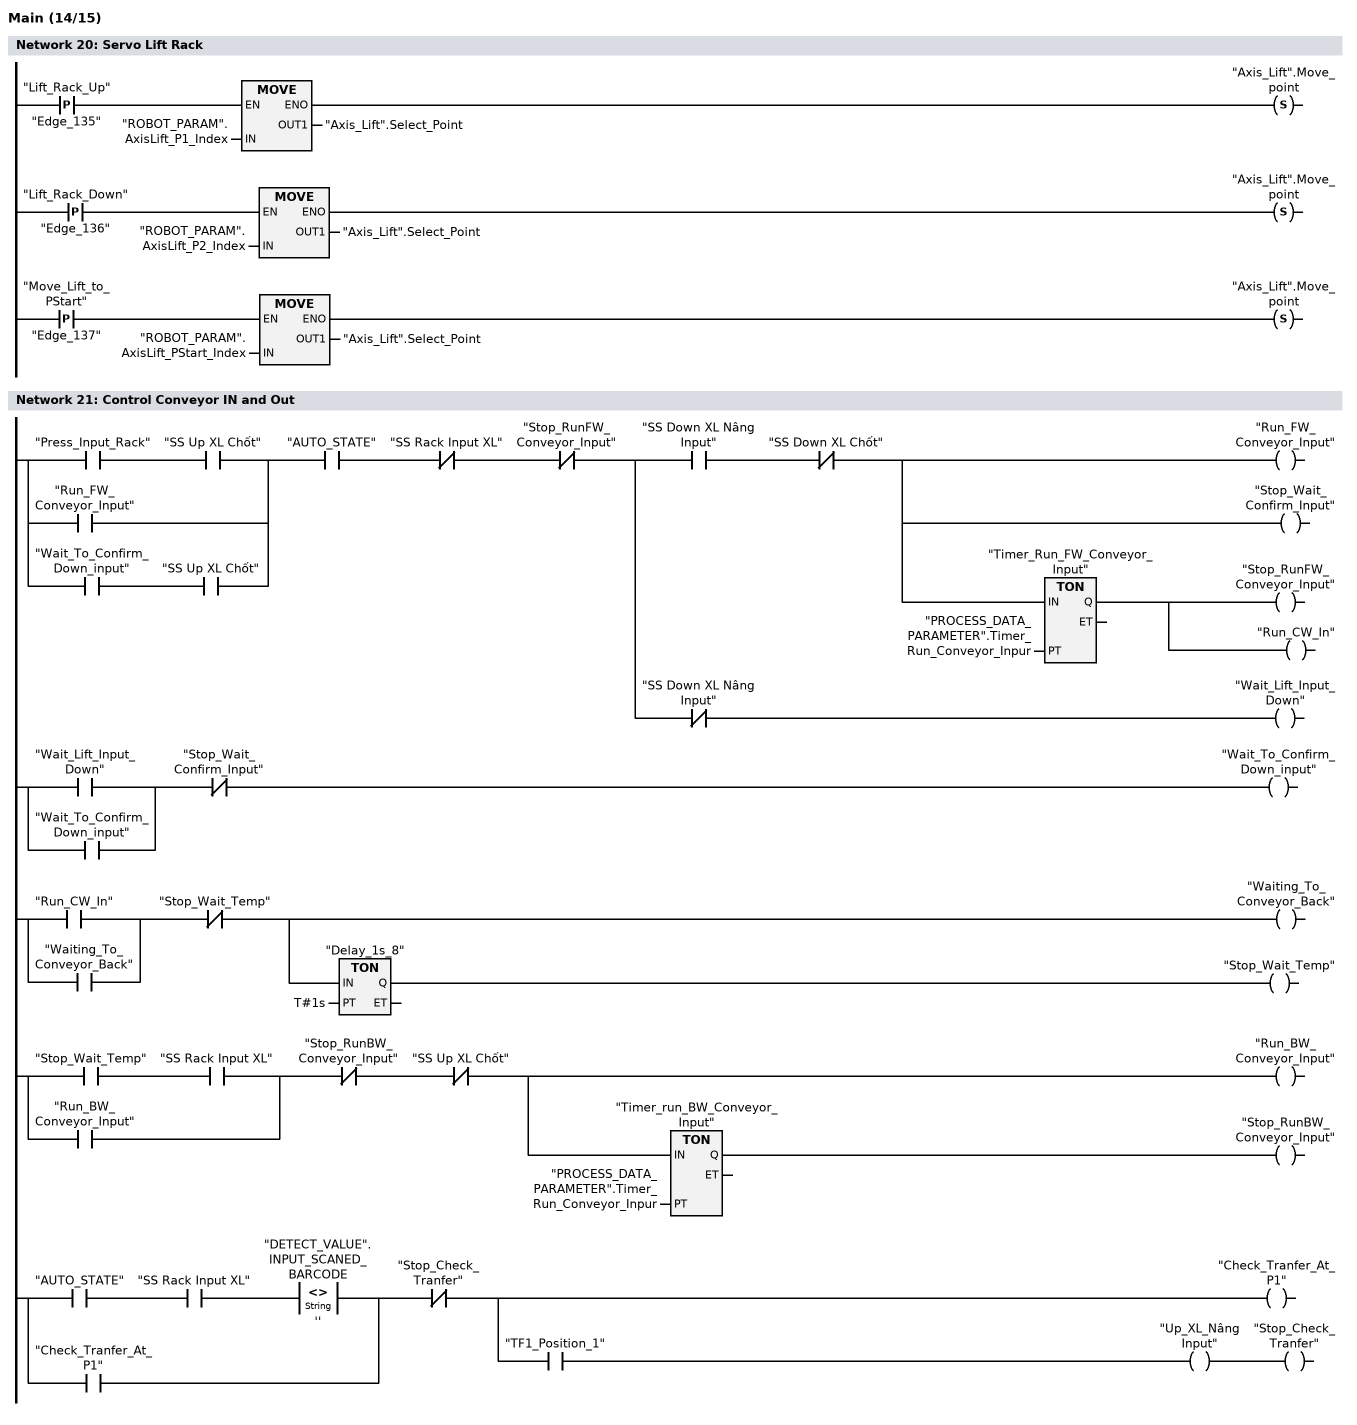
   RUNG wire#powerrail
      P_Contact(operand := "Lift_Rack_Up", bit := "Edge_135")
      { S7_GenerateENO := "TRUE" } Move(in := "ROBOT_PARAM".AxisLift_P1_Index, out1 => "Axis_Lift".Select_Point)
      S_Coil( "Axis_Lift".Move_point )
   END_RUNG
   RUNG wire#powerrail
      P_Contact(operand := "Lift_Rack_Down", bit := "Edge_136")
      { S7_GenerateENO := "TRUE" } Move(in := "ROBOT_PARAM".AxisLift_P2_Index, out1 => "Axis_Lift".Select_Point)
      S_Coil( "Axis_Lift".Move_point )
   END_RUNG
   RUNG wire#powerrail
      P_Contact(operand := "Move_Lift_to_PStart", bit := "Edge_137")
      { S7_GenerateENO := "TRUE" } Move(in := "ROBOT_PARAM".AxisLift_PStart_Index, out1 => "Axis_Lift".Select_Point)
      S_Coil( "Axis_Lift".Move_point )
   END_RUNG
   // the same network as SCL:
   // ENO of a box is taken as its EN; it also drops when the box reports an error
   #_w1 := "Lift_Rack_Up" AND NOT "Edge_135";   // rising edge of "Lift_Rack_Up"
   "Edge_135" := "Lift_Rack_Up";
   IF #_w1 THEN
       "Axis_Lift".Select_Point := "ROBOT_PARAM".AxisLift_P1_Index;
       "Axis_Lift".Move_point := TRUE;
   END_IF;
   #_w2 := "Lift_Rack_Down" AND NOT "Edge_136";   // rising edge of "Lift_Rack_Down"
   "Edge_136" := "Lift_Rack_Down";
   IF #_w2 THEN
       "Axis_Lift".Select_Point := "ROBOT_PARAM".AxisLift_P2_Index;
       "Axis_Lift".Move_point := TRUE;
   END_IF;
   #_w3 := "Move_Lift_to_PStart" AND NOT "Edge_137";   // rising edge of "Move_Lift_to_PStart"
   "Edge_137" := "Move_Lift_to_PStart";
   IF #_w3 THEN
       "Axis_Lift".Select_Point := "ROBOT_PARAM".AxisLift_PStart_Index;
       "Axis_Lift".Move_point := TRUE;
   END_IF;
END_REGION

REGION Network 21: Control Conveyor IN and Out
   #_w1 := (("Press_Input_Rack" AND "SS Up XL Chốt") OR "Run_FW_Conveyor_Input" OR ("Wait_To_Confirm_Down_input" AND "SS Up XL Chốt")) AND "AUTO_STATE" AND NOT "SS Rack Input XL" AND NOT "Stop_RunFW_Conveyor_Input";
   "Run_FW_Conveyor_Input" := #_w1 AND "SS Down XL Nâng Input" AND NOT "SS Down XL Chốt";
   "Stop_Wait_Confirm_Input" := "Run_FW_Conveyor_Input";
   "Timer_Run_FW_Conveyor_Input".TON(IN := "Run_FW_Conveyor_Input",
                           PT := "PROCESS_DATA_PARAMETER".Timer_Run_Conveyor_Inpur);
   "Stop_RunFW_Conveyor_Input" := "Timer_Run_FW_Conveyor_Input".Q;
   "Run_CW_In" := "Timer_Run_FW_Conveyor_Input".Q;
   "Wait_Lift_Input_Down" := #_w1 AND NOT "SS Down XL Nâng Input";
   "Wait_To_Confirm_Down_input" := ("Wait_Lift_Input_Down" OR "Wait_To_Confirm_Down_input") AND NOT "Stop_Wait_Confirm_Input";
   "Waiting_To_Conveyor_Back" := ("Run_CW_In" OR "Waiting_To_Conveyor_Back") AND NOT "Stop_Wait_Temp";
   "Delay_1s_8".TON(IN := "Waiting_To_Conveyor_Back", PT := T#1s);
   "Stop_Wait_Temp" := "Delay_1s_8".Q;
   "Run_BW_Conveyor_Input" := (("Stop_Wait_Temp" AND "SS Rack Input XL") OR "Run_BW_Conveyor_Input") AND NOT "Stop_RunBW_Conveyor_Input" AND NOT "SS Up XL Chốt";
   "Timer_run_BW_Conveyor_Input".TON(IN := "Run_BW_Conveyor_Input",
                           PT := "PROCESS_DATA_PARAMETER".Timer_Run_Conveyor_Inpur);
   "Stop_RunBW_Conveyor_Input" := "Timer_run_BW_Conveyor_Input".Q;
   "Check_Tranfer_At_P1" := (("AUTO_STATE" AND "SS Rack Input XL" AND ("DETECT_VALUE".INPUT_SCANED_BARCODE <> '')) OR "Check_Tranfer_At_P1") AND NOT "Stop_Check_Tranfer";
   "Up_XL_Nâng Input" := "Check_Tranfer_At_P1" AND "TF1_Position_1";
   "Stop_Check_Tranfer" := "Up_XL_Nâng Input";
END_REGION

REGION Network 22: Conveyor Out
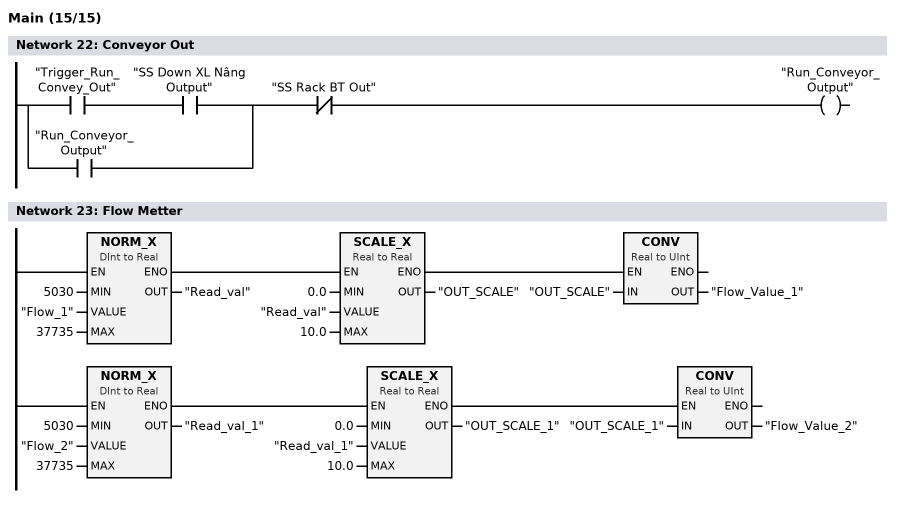
   RUNG wire#powerrail
      Contact( "Trigger_Run_Convey_Out" )
      Contact( "SS Down XL Nâng Output" )
      wire#w1
      I_Contact( "SS Rack BT Out" )
      Coil( "Run_Conveyor_Output" )
   END_RUNG
   RUNG wire#powerrail
      Contact( "Run_Conveyor_Output" )
   END_RUNG wire#w1
   // the same network as SCL:
   "Run_Conveyor_Output" := (("Trigger_Run_Convey_Out" AND "SS Down XL Nâng Output") OR "Run_Conveyor_Output") AND NOT "SS Rack BT Out";
END_REGION

REGION Network 23: Flow Metter
   RUNG wire#powerrail
      { S7_Templates := "[SrcType := DInt, DestType := Real]"; S7_GenerateENO := "TRUE" } Normalize(min := 5030, value := "Flow_1", max := 37735, out => "Read_val")
      { S7_Templates := "[SrcType := Real, DestType := Real]"; S7_GenerateENO := "TRUE" } Scale(min := 0.0, value := "Read_val", max := 10.0, out => "OUT_SCALE")
      { S7_Templates := "[SrcType := Real, DestType := UInt]"; S7_GenerateENO := "TRUE" } Convert(in := "OUT_SCALE", out => "Flow_Value_1")
   END_RUNG
   RUNG wire#powerrail
      { S7_Templates := "[SrcType := DInt, DestType := Real]"; S7_GenerateENO := "TRUE" } Normalize(min := 5030, value := "Flow_2", max := 37735, out => "Read_val_1")
      { S7_Templates := "[SrcType := Real, DestType := Real]"; S7_GenerateENO := "TRUE" } Scale(min := 0.0, value := "Read_val_1", max := 10.0, out => "OUT_SCALE_1")
      { S7_Templates := "[SrcType := Real, DestType := UInt]"; S7_GenerateENO := "TRUE" } Convert(in := "OUT_SCALE_1", out => "Flow_Value_2")
   END_RUNG
   // the same network as SCL:
   // ENO of a box is taken as its EN; it also drops when the box reports an error
   "Read_val" := NORM_X(MIN := 5030, VALUE := "Flow_1", MAX := 37735);
   "OUT_SCALE" := SCALE_X(MIN := 0.0, VALUE := "Read_val", MAX := 10.0);
   "Flow_Value_1" := REAL_TO_UINT("OUT_SCALE");
   "Read_val_1" := NORM_X(MIN := 5030, VALUE := "Flow_2", MAX := 37735);
   "OUT_SCALE_1" := SCALE_X(MIN := 0.0, VALUE := "Read_val_1", MAX := 10.0);
   "Flow_Value_2" := REAL_TO_UINT("OUT_SCALE_1");
END_REGION
END_ORGANIZATION_BLOCK

ORGANIZATION_BLOCK "MOTOR_CONTROL"   // OB123, LAD, ProgramCycle
TITLE = "Main Program Sweep (Cycle)"
{ S7_Optimized_Access := 'TRUE' }
VERSION : 0.1
   VAR_INPUT
      Initial_Call : Bool;   // Initial call of this OB
      Remanence : Bool;   // =True, if remanent data are available
   END_VAR
   VAR_TEMP   // added for the SCL form of the ladder/FBD networks
      _w1 : Bool;
      _w2 : Bool;
      _w3 : Bool;
      _w4 : Bool;
      _w5 : Bool;
      _w6 : Bool;
      _w7 : Bool;
      _w8 : Bool;
      _w9 : Bool;
      _w10 : Bool;
      _w11 : Bool;
      _w12 : Bool;
      _w13 : Bool;
      _w14 : Bool;
      _w15 : Bool;
      _w16 : Bool;
      _w17 : Bool;
      _w18 : Bool;
      _w19 : Bool;
      _w20 : Bool;
      _w21 : Bool;
      _w22 : Bool;
      _w23 : Bool;
      _w24 : Bool;
      _w25 : Bool;
      _w26 : Bool;
      _w27 : Bool;
      _w28 : Bool;
      _w29 : Bool;
      _w30 : Bool;
      _w31 : Bool;
      _w32 : Bool;
      _w33 : Bool;
      _w34 : Bool;
      _w35 : Bool;
      _w36 : Bool;
      _w37 : Bool;
      _w38 : Bool;
      _w39 : Bool;
      _w40 : Bool;
   END_VAR
BEGIN

REGION Network 1: MODBUS INITIALIZE
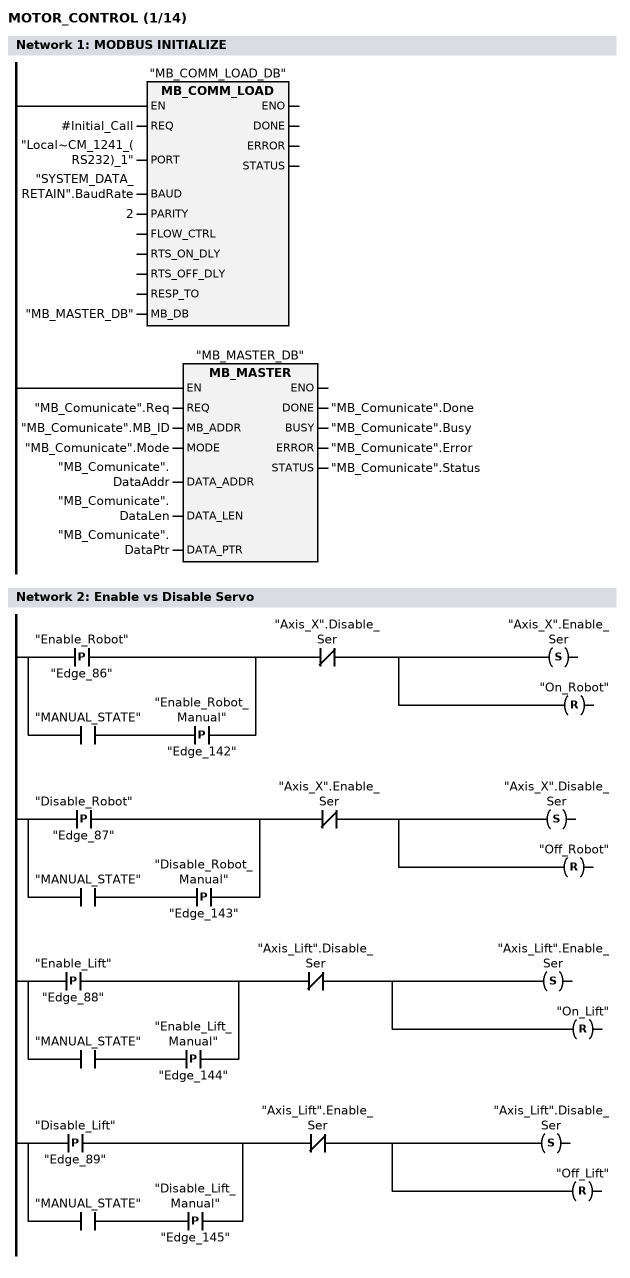
   "MB_COMM_LOAD_DB"(REQ := #Initial_Call,   // MB_COMM_LOAD
                     PORT := "Local~CM_1241_(RS232)_1",
                     BAUD := "SYSTEM_DATA_RETAIN".BaudRate,
                     PARITY := 2,
                     MB_DB := "MB_MASTER_DB");
   "MB_MASTER_DB"(REQ := "MB_Comunicate".Req,   // MB_MASTER
                  MB_ADDR := "MB_Comunicate".MB_ID,
                  MODE := "MB_Comunicate".Mode,
                  DATA_ADDR := "MB_Comunicate".DataAddr,
                  DATA_LEN := "MB_Comunicate".DataLen,
                  DATA_PTR := "MB_Comunicate".DataPtr,
                  DONE => "MB_Comunicate".Done,
                  BUSY => "MB_Comunicate".Busy,
                  ERROR => "MB_Comunicate".Error,
                  STATUS => "MB_Comunicate".Status);
END_REGION

REGION Network 2: Enable vs Disable Servo
   RUNG wire#powerrail
      P_Contact(operand := "Enable_Robot", bit := "Edge_86")
      wire#w1
      I_Contact( "Axis_X".Disable_Ser )
      wire#w2
      S_Coil( "Axis_X".Enable_Ser )
   END_RUNG
   RUNG wire#powerrail
      Contact( "MANUAL_STATE" )
      P_Contact(operand := "Enable_Robot_Manual", bit := "Edge_142")
   END_RUNG wire#w1
   RUNG wire#w2
      R_Coil( "On_Robot" )
   END_RUNG
   RUNG wire#powerrail
      P_Contact(operand := "Disable_Robot", bit := "Edge_87")
      wire#w3
      I_Contact( "Axis_X".Enable_Ser )
      wire#w4
      S_Coil( "Axis_X".Disable_Ser )
   END_RUNG
   RUNG wire#powerrail
      Contact( "MANUAL_STATE" )
      P_Contact(operand := "Disable_Robot_Manual", bit := "Edge_143")
   END_RUNG wire#w3
   RUNG wire#w4
      R_Coil( "Off_Robot" )
   END_RUNG
   RUNG wire#powerrail
      P_Contact(operand := "Enable_Lift", bit := "Edge_88")
      wire#w5
      I_Contact( "Axis_Lift".Disable_Ser )
      wire#w6
      S_Coil( "Axis_Lift".Enable_Ser )
   END_RUNG
   RUNG wire#powerrail
      Contact( "MANUAL_STATE" )
      P_Contact(operand := "Enable_Lift_Manual", bit := "Edge_144")
   END_RUNG wire#w5
   RUNG wire#w6
      R_Coil( "On_Lift" )
   END_RUNG
   RUNG wire#powerrail
      P_Contact(operand := "Disable_Lift", bit := "Edge_89")
      wire#w7
      I_Contact( "Axis_Lift".Enable_Ser )
      wire#w8
      S_Coil( "Axis_Lift".Disable_Ser )
   END_RUNG
   RUNG wire#powerrail
      Contact( "MANUAL_STATE" )
      P_Contact(operand := "Disable_Lift_Manual", bit := "Edge_145")
   END_RUNG wire#w7
   RUNG wire#w8
      R_Coil( "Off_Lift" )
   END_RUNG
   // the same network as SCL:
   #_w1 := "Enable_Robot" AND NOT "Edge_86";   // rising edge of "Enable_Robot"
   "Edge_86" := "Enable_Robot";
   #_w2 := "MANUAL_STATE" AND "Enable_Robot_Manual" AND NOT "Edge_142";   // rising edge of "Enable_Robot_Manual"
   "Edge_142" := "Enable_Robot_Manual";
   IF (#_w1 OR #_w2) AND NOT "Axis_X".Disable_Ser THEN
       "Axis_X".Enable_Ser := TRUE;
       "On_Robot" := FALSE;
   END_IF;
   #_w3 := "Disable_Robot" AND NOT "Edge_87";   // rising edge of "Disable_Robot"
   "Edge_87" := "Disable_Robot";
   #_w4 := "MANUAL_STATE" AND "Disable_Robot_Manual" AND NOT "Edge_143";   // rising edge of "Disable_Robot_Manual"
   "Edge_143" := "Disable_Robot_Manual";
   IF (#_w3 OR #_w4) AND NOT "Axis_X".Enable_Ser THEN
       "Axis_X".Disable_Ser := TRUE;
       "Off_Robot" := FALSE;
   END_IF;
   #_w5 := "Enable_Lift" AND NOT "Edge_88";   // rising edge of "Enable_Lift"
   "Edge_88" := "Enable_Lift";
   #_w6 := "MANUAL_STATE" AND "Enable_Lift_Manual" AND NOT "Edge_144";   // rising edge of "Enable_Lift_Manual"
   "Edge_144" := "Enable_Lift_Manual";
   IF (#_w5 OR #_w6) AND NOT "Axis_Lift".Disable_Ser THEN
       "Axis_Lift".Enable_Ser := TRUE;
       "On_Lift" := FALSE;
   END_IF;
   #_w7 := "Disable_Lift" AND NOT "Edge_89";   // rising edge of "Disable_Lift"
   "Edge_89" := "Disable_Lift";
   #_w8 := "MANUAL_STATE" AND "Disable_Lift_Manual" AND NOT "Edge_145";   // rising edge of "Disable_Lift_Manual"
   "Edge_145" := "Disable_Lift_Manual";
   IF (#_w7 OR #_w8) AND NOT "Axis_Lift".Enable_Ser THEN
       "Axis_Lift".Disable_Ser := TRUE;
       "Off_Lift" := FALSE;
   END_IF;
END_REGION

REGION Network 3: AXIS X
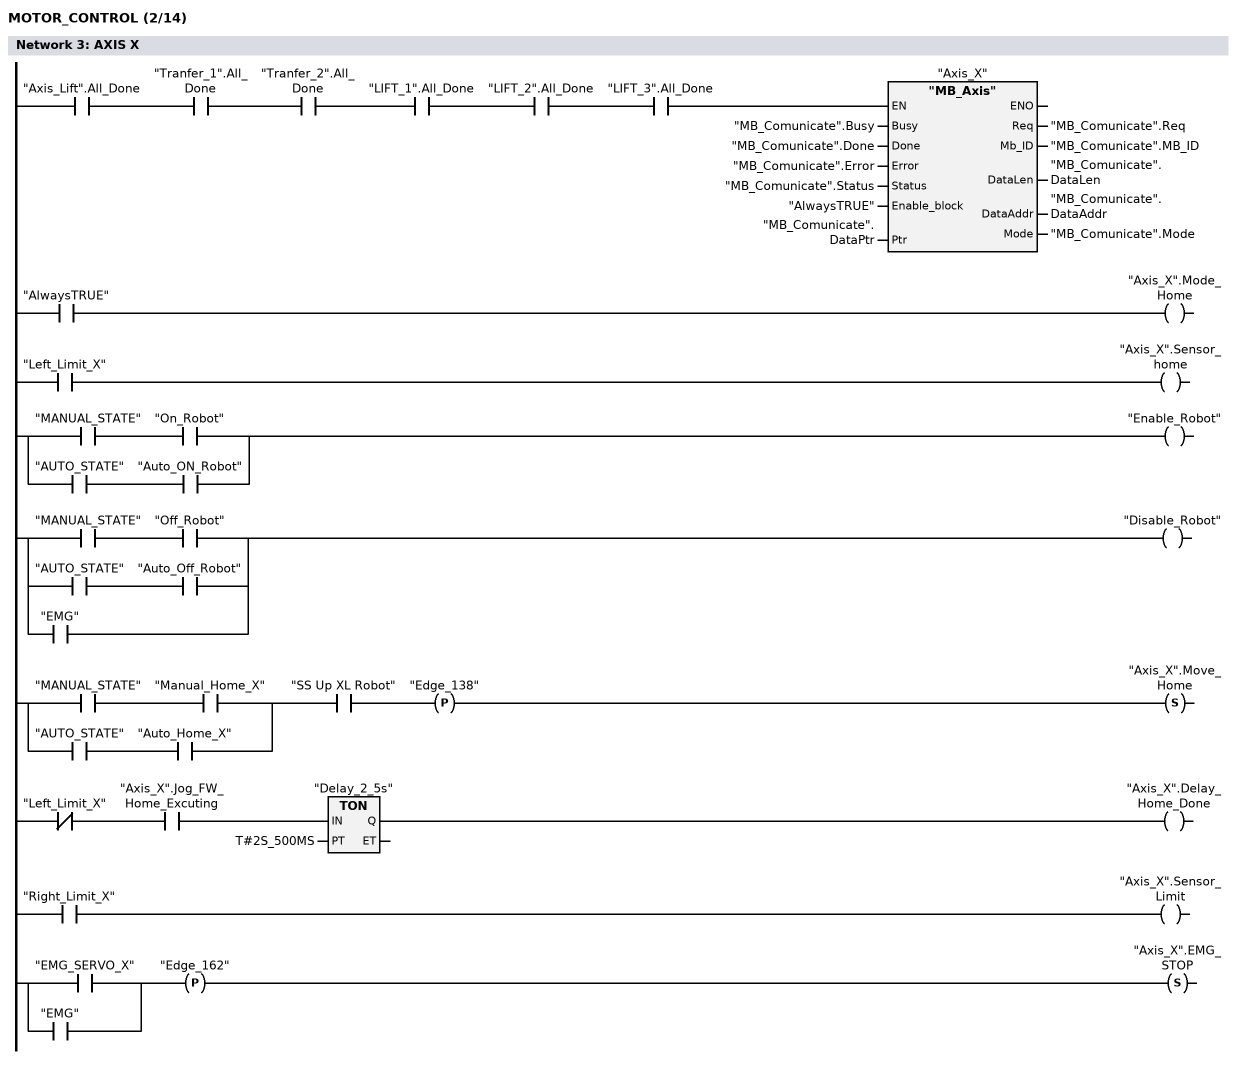
   IF "Axis_Lift".All_Done AND "Tranfer_1".All_Done AND "Tranfer_2".All_Done AND "LIFT_1".All_Done AND "LIFT_2".All_Done AND "LIFT_3".All_Done THEN
       "Axis_X"(Busy := "MB_Comunicate".Busy,   // "MB_Axis"
                Done := "MB_Comunicate".Done,
                Error := "MB_Comunicate".Error,
                Status := "MB_Comunicate".Status,
                Enable_block := "AlwaysTRUE",
                Ptr := "MB_Comunicate".DataPtr,
                Req => "MB_Comunicate".Req,
                Mb_ID => "MB_Comunicate".MB_ID,
                DataLen => "MB_Comunicate".DataLen,
                DataAddr => "MB_Comunicate".DataAddr,
                Mode => "MB_Comunicate".Mode);
   END_IF;
   "Axis_X".Mode_Home := "AlwaysTRUE";
   "Axis_X".Sensor_home := "Left_Limit_X";
   "Enable_Robot" := ("MANUAL_STATE" AND "On_Robot") OR ("AUTO_STATE" AND "Auto_ON_Robot");
   "Disable_Robot" := ("MANUAL_STATE" AND "Off_Robot") OR ("AUTO_STATE" AND "Auto_Off_Robot") OR "EMG";
   #_w1 := (("MANUAL_STATE" AND "Manual_Home_X") OR ("AUTO_STATE" AND "Auto_Home_X")) AND "SS Up XL Robot";
   #_w2 := #_w1 AND NOT "Edge_138";   // rising edge
   "Edge_138" := #_w1;
   IF #_w2 THEN "Axis_X".Move_Home := TRUE; END_IF;
   "Delay_2_5s".TON(IN := NOT "Left_Limit_X" AND "Axis_X".Jog_FW_Home_Excuting, PT := T#2S_500MS);
   "Axis_X".Delay_Home_Done := "Delay_2_5s".Q;
   "Axis_X".Sensor_Limit := "Right_Limit_X";
   #_w3 := "EMG_SERVO_X" OR "EMG";
   #_w4 := #_w3 AND NOT "Edge_162";   // rising edge
   "Edge_162" := #_w3;
   IF #_w4 THEN "Axis_X".EMG_STOP := TRUE; END_IF;
END_REGION

REGION Network 4: AXIS LIFT
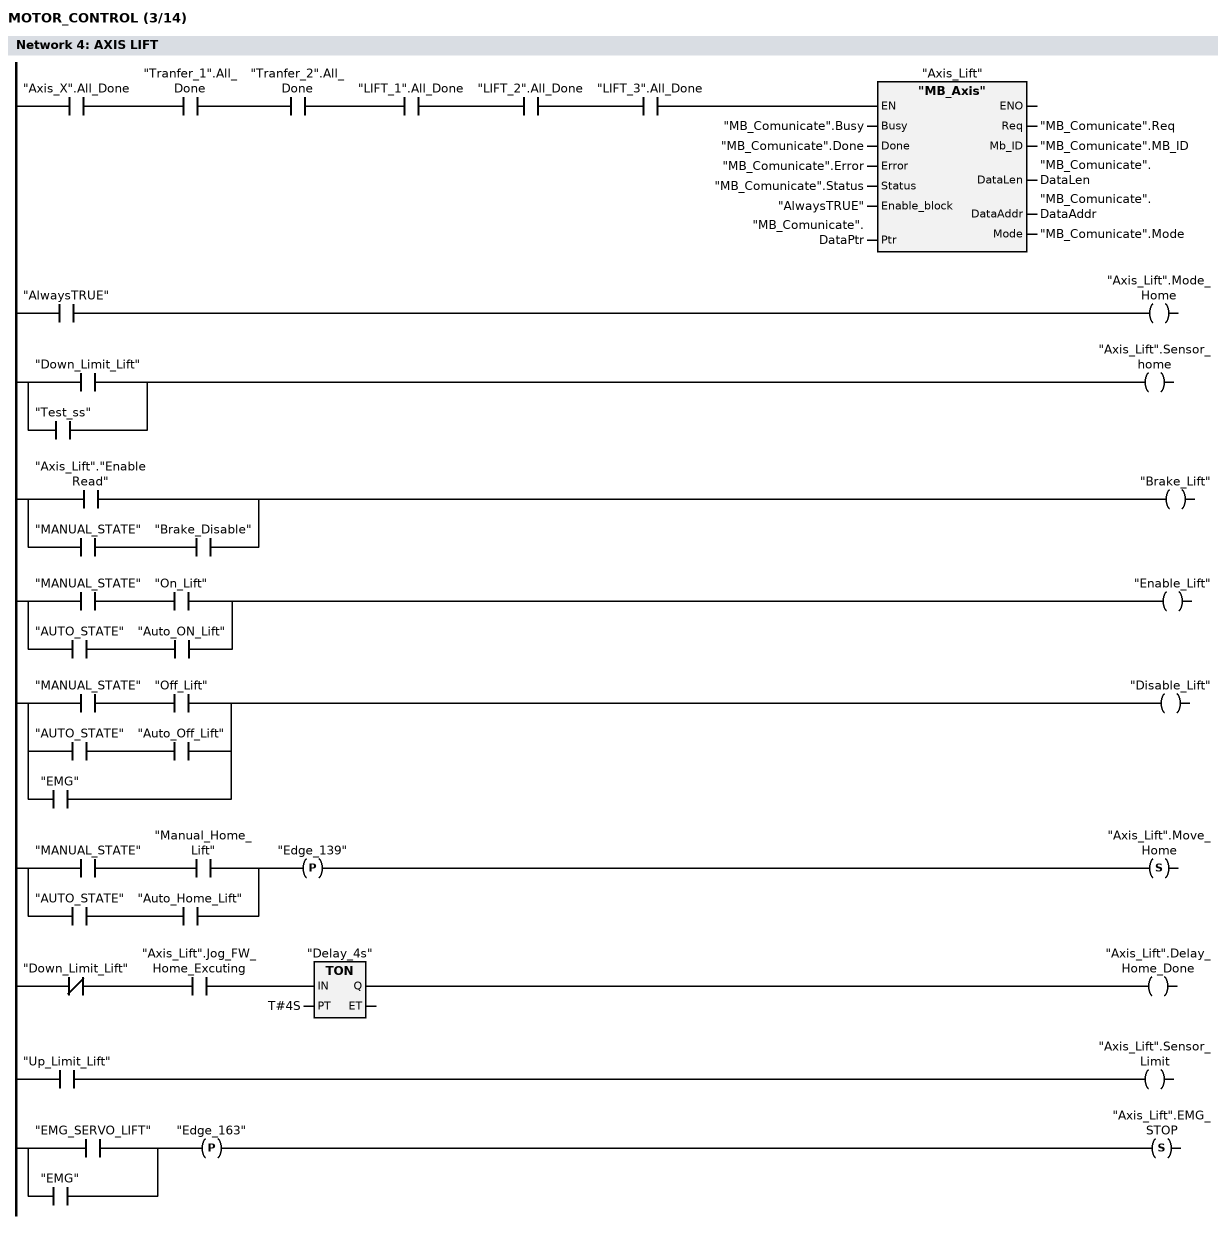
   IF "Axis_X".All_Done AND "Tranfer_1".All_Done AND "Tranfer_2".All_Done AND "LIFT_1".All_Done AND "LIFT_2".All_Done AND "LIFT_3".All_Done THEN
       "Axis_Lift"(Busy := "MB_Comunicate".Busy,   // "MB_Axis"
                   Done := "MB_Comunicate".Done,
                   Error := "MB_Comunicate".Error,
                   Status := "MB_Comunicate".Status,
                   Enable_block := "AlwaysTRUE",
                   Ptr := "MB_Comunicate".DataPtr,
                   Req => "MB_Comunicate".Req,
                   Mb_ID => "MB_Comunicate".MB_ID,
                   DataLen => "MB_Comunicate".DataLen,
                   DataAddr => "MB_Comunicate".DataAddr,
                   Mode => "MB_Comunicate".Mode);
   END_IF;
   "Axis_Lift".Mode_Home := "AlwaysTRUE";
   "Axis_Lift".Sensor_home := "Down_Limit_Lift" OR "Test_ss";
   "Brake_Lift" := "Axis_Lift"."Enable Read" OR ("MANUAL_STATE" AND "Brake_Disable");
   "Enable_Lift" := ("MANUAL_STATE" AND "On_Lift") OR ("AUTO_STATE" AND "Auto_ON_Lift");
   "Disable_Lift" := ("MANUAL_STATE" AND "Off_Lift") OR ("AUTO_STATE" AND "Auto_Off_Lift") OR "EMG";
   #_w1 := ("MANUAL_STATE" AND "Manual_Home_Lift") OR ("AUTO_STATE" AND "Auto_Home_Lift");
   #_w2 := #_w1 AND NOT "Edge_139";   // rising edge
   "Edge_139" := #_w1;
   IF #_w2 THEN "Axis_Lift".Move_Home := TRUE; END_IF;
   "Delay_4s".TON(IN := NOT "Down_Limit_Lift" AND "Axis_Lift".Jog_FW_Home_Excuting, PT := T#4S);
   "Axis_Lift".Delay_Home_Done := "Delay_4s".Q;
   "Axis_Lift".Sensor_Limit := "Up_Limit_Lift";
   #_w3 := "EMG_SERVO_LIFT" OR "EMG";
   #_w4 := #_w3 AND NOT "Edge_163";   // rising edge
   "Edge_163" := #_w3;
   IF #_w4 THEN "Axis_Lift".EMG_STOP := TRUE; END_IF;
END_REGION

REGION Network 5: Data Position
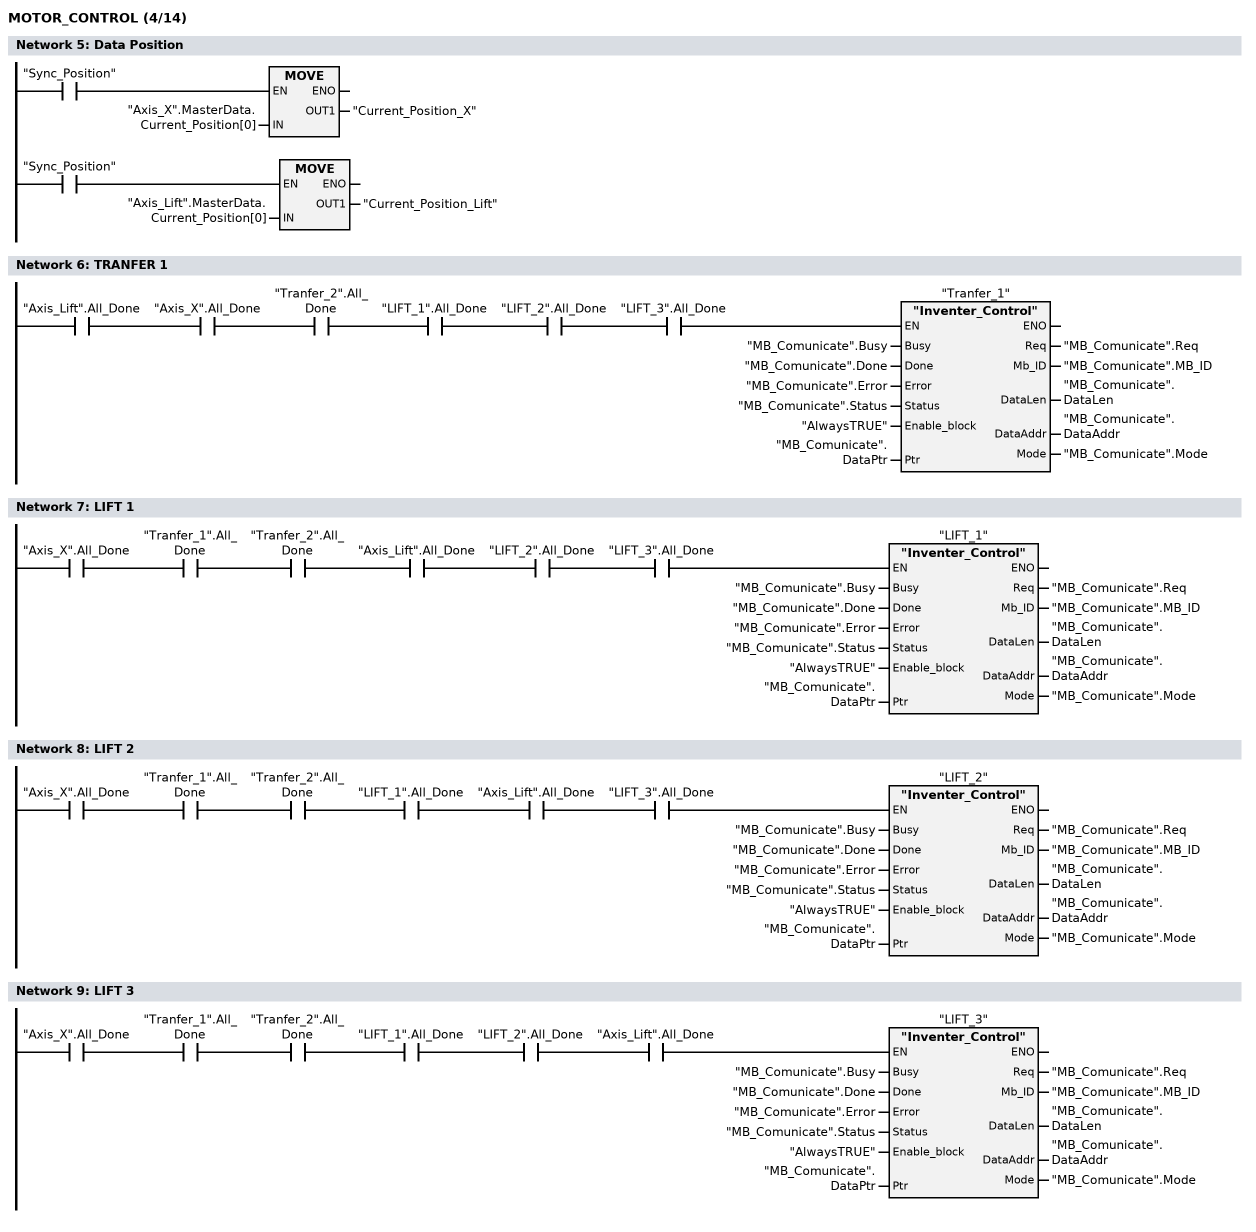
   RUNG wire#powerrail
      Contact( "Sync_Position" )
      { S7_GenerateENO := "TRUE" } Move(in := "Axis_X".MasterData.Current_Position[0], out1 => "Current_Position_X")
   END_RUNG
   RUNG wire#powerrail
      Contact( "Sync_Position" )
      { S7_GenerateENO := "TRUE" } Move(in := "Axis_Lift".MasterData.Current_Position[0], out1 => "Current_Position_Lift")
   END_RUNG
   // the same network as SCL:
   IF "Sync_Position" THEN
       "Current_Position_X" := "Axis_X".MasterData.Current_Position[0];
       "Current_Position_Lift" := "Axis_Lift".MasterData.Current_Position[0];
   END_IF;
END_REGION

REGION Network 6: TRANFER 1
   RUNG wire#powerrail
      Contact( "Axis_Lift".All_Done )
      Contact( "Axis_X".All_Done )
      Contact( "Tranfer_2".All_Done )
      Contact( "LIFT_1".All_Done )
      Contact( "LIFT_2".All_Done )
      Contact( "LIFT_3".All_Done )
      "Tranfer_1"(Busy := "MB_Comunicate".Busy, Done := "MB_Comunicate".Done, Error := "MB_Comunicate".Error, Status := "MB_Comunicate".Status, Enable_block := "AlwaysTRUE", Ptr := "MB_Comunicate".DataPtr, Req => "MB_Comunicate".Req, Mb_ID => "MB_Comunicate".MB_ID, DataLen => "MB_Comunicate".DataLen, DataAddr => "MB_Comunicate".DataAddr, Mode => "MB_Comunicate".Mode)
   END_RUNG
   // the same network as SCL:
   IF "Axis_Lift".All_Done AND "Axis_X".All_Done AND "Tranfer_2".All_Done AND "LIFT_1".All_Done AND "LIFT_2".All_Done AND "LIFT_3".All_Done THEN
       "Tranfer_1"(Busy := "MB_Comunicate".Busy,   // "Inventer_Control"
                   Done := "MB_Comunicate".Done,
                   Error := "MB_Comunicate".Error,
                   Status := "MB_Comunicate".Status,
                   Enable_block := "AlwaysTRUE",
                   Ptr := "MB_Comunicate".DataPtr,
                   Req => "MB_Comunicate".Req,
                   Mb_ID => "MB_Comunicate".MB_ID,
                   DataLen => "MB_Comunicate".DataLen,
                   DataAddr => "MB_Comunicate".DataAddr,
                   Mode => "MB_Comunicate".Mode);
   END_IF;
END_REGION

REGION Network 7: LIFT 1
   RUNG wire#powerrail
      Contact( "Axis_X".All_Done )
      Contact( "Tranfer_1".All_Done )
      Contact( "Tranfer_2".All_Done )
      Contact( "Axis_Lift".All_Done )
      Contact( "LIFT_2".All_Done )
      Contact( "LIFT_3".All_Done )
      "LIFT_1"(Busy := "MB_Comunicate".Busy, Done := "MB_Comunicate".Done, Error := "MB_Comunicate".Error, Status := "MB_Comunicate".Status, Enable_block := "AlwaysTRUE", Ptr := "MB_Comunicate".DataPtr, Req => "MB_Comunicate".Req, Mb_ID => "MB_Comunicate".MB_ID, DataLen => "MB_Comunicate".DataLen, DataAddr => "MB_Comunicate".DataAddr, Mode => "MB_Comunicate".Mode)
   END_RUNG
   // the same network as SCL:
   IF "Axis_X".All_Done AND "Tranfer_1".All_Done AND "Tranfer_2".All_Done AND "Axis_Lift".All_Done AND "LIFT_2".All_Done AND "LIFT_3".All_Done THEN
       "LIFT_1"(Busy := "MB_Comunicate".Busy,   // "Inventer_Control"
                Done := "MB_Comunicate".Done,
                Error := "MB_Comunicate".Error,
                Status := "MB_Comunicate".Status,
                Enable_block := "AlwaysTRUE",
                Ptr := "MB_Comunicate".DataPtr,
                Req => "MB_Comunicate".Req,
                Mb_ID => "MB_Comunicate".MB_ID,
                DataLen => "MB_Comunicate".DataLen,
                DataAddr => "MB_Comunicate".DataAddr,
                Mode => "MB_Comunicate".Mode);
   END_IF;
END_REGION

REGION Network 8: LIFT 2
   RUNG wire#powerrail
      Contact( "Axis_X".All_Done )
      Contact( "Tranfer_1".All_Done )
      Contact( "Tranfer_2".All_Done )
      Contact( "LIFT_1".All_Done )
      Contact( "Axis_Lift".All_Done )
      Contact( "LIFT_3".All_Done )
      "LIFT_2"(Busy := "MB_Comunicate".Busy, Done := "MB_Comunicate".Done, Error := "MB_Comunicate".Error, Status := "MB_Comunicate".Status, Enable_block := "AlwaysTRUE", Ptr := "MB_Comunicate".DataPtr, Req => "MB_Comunicate".Req, Mb_ID => "MB_Comunicate".MB_ID, DataLen => "MB_Comunicate".DataLen, DataAddr => "MB_Comunicate".DataAddr, Mode => "MB_Comunicate".Mode)
   END_RUNG
   // the same network as SCL:
   IF "Axis_X".All_Done AND "Tranfer_1".All_Done AND "Tranfer_2".All_Done AND "LIFT_1".All_Done AND "Axis_Lift".All_Done AND "LIFT_3".All_Done THEN
       "LIFT_2"(Busy := "MB_Comunicate".Busy,   // "Inventer_Control"
                Done := "MB_Comunicate".Done,
                Error := "MB_Comunicate".Error,
                Status := "MB_Comunicate".Status,
                Enable_block := "AlwaysTRUE",
                Ptr := "MB_Comunicate".DataPtr,
                Req => "MB_Comunicate".Req,
                Mb_ID => "MB_Comunicate".MB_ID,
                DataLen => "MB_Comunicate".DataLen,
                DataAddr => "MB_Comunicate".DataAddr,
                Mode => "MB_Comunicate".Mode);
   END_IF;
END_REGION

REGION Network 9: LIFT 3
   RUNG wire#powerrail
      Contact( "Axis_X".All_Done )
      Contact( "Tranfer_1".All_Done )
      Contact( "Tranfer_2".All_Done )
      Contact( "LIFT_1".All_Done )
      Contact( "LIFT_2".All_Done )
      Contact( "Axis_Lift".All_Done )
      "LIFT_3"(Busy := "MB_Comunicate".Busy, Done := "MB_Comunicate".Done, Error := "MB_Comunicate".Error, Status := "MB_Comunicate".Status, Enable_block := "AlwaysTRUE", Ptr := "MB_Comunicate".DataPtr, Req => "MB_Comunicate".Req, Mb_ID => "MB_Comunicate".MB_ID, DataLen => "MB_Comunicate".DataLen, DataAddr => "MB_Comunicate".DataAddr, Mode => "MB_Comunicate".Mode)
   END_RUNG
   // the same network as SCL:
   IF "Axis_X".All_Done AND "Tranfer_1".All_Done AND "Tranfer_2".All_Done AND "LIFT_1".All_Done AND "LIFT_2".All_Done AND "Axis_Lift".All_Done THEN
       "LIFT_3"(Busy := "MB_Comunicate".Busy,   // "Inventer_Control"
                Done := "MB_Comunicate".Done,
                Error := "MB_Comunicate".Error,
                Status := "MB_Comunicate".Status,
                Enable_block := "AlwaysTRUE",
                Ptr := "MB_Comunicate".DataPtr,
                Req => "MB_Comunicate".Req,
                Mb_ID => "MB_Comunicate".MB_ID,
                DataLen => "MB_Comunicate".DataLen,
                DataAddr => "MB_Comunicate".DataAddr,
                Mode => "MB_Comunicate".Mode);
   END_IF;
END_REGION

REGION Network 10
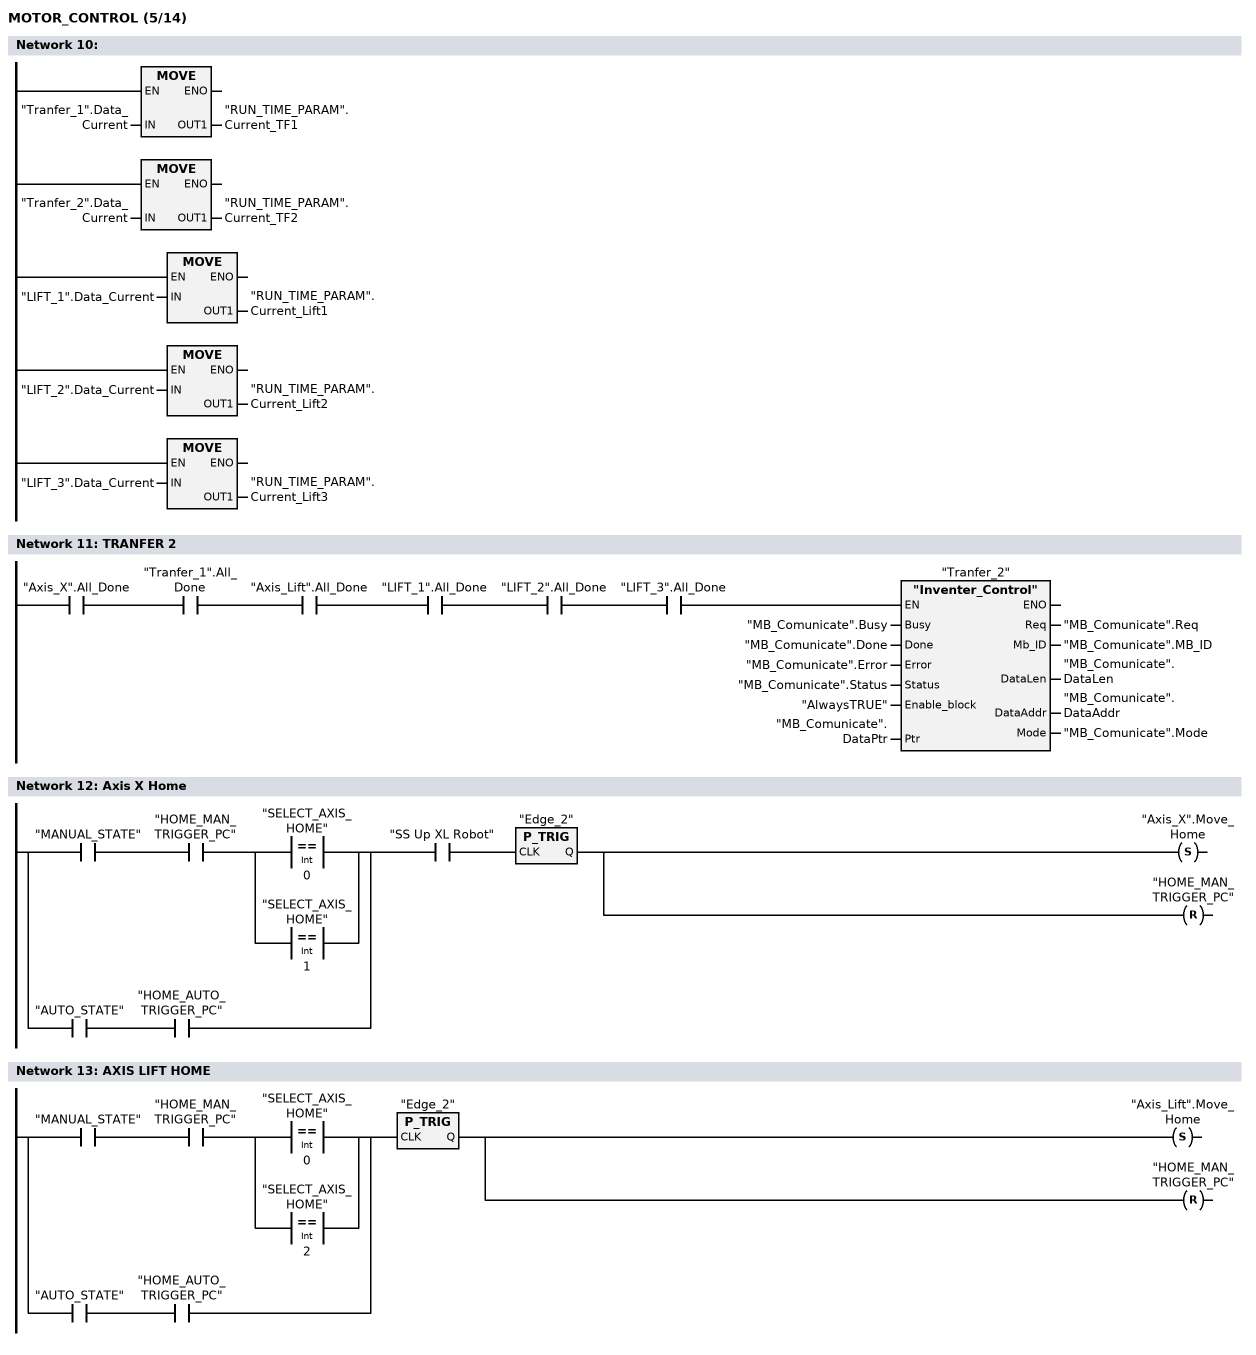
   RUNG wire#powerrail
      { S7_GenerateENO := "TRUE" } Move(in := "Tranfer_1".Data_Current, out1 => "RUN_TIME_PARAM".Current_TF1)
   END_RUNG
   RUNG wire#powerrail
      { S7_GenerateENO := "TRUE" } Move(in := "Tranfer_2".Data_Current, out1 => "RUN_TIME_PARAM".Current_TF2)
   END_RUNG
   RUNG wire#powerrail
      { S7_GenerateENO := "TRUE" } Move(in := "LIFT_1".Data_Current, out1 => "RUN_TIME_PARAM".Current_Lift1)
   END_RUNG
   RUNG wire#powerrail
      { S7_GenerateENO := "TRUE" } Move(in := "LIFT_2".Data_Current, out1 => "RUN_TIME_PARAM".Current_Lift2)
   END_RUNG
   RUNG wire#powerrail
      { S7_GenerateENO := "TRUE" } Move(in := "LIFT_3".Data_Current, out1 => "RUN_TIME_PARAM".Current_Lift3)
   END_RUNG
   // the same network as SCL:
   "RUN_TIME_PARAM".Current_TF1 := "Tranfer_1".Data_Current;
   "RUN_TIME_PARAM".Current_TF2 := "Tranfer_2".Data_Current;
   "RUN_TIME_PARAM".Current_Lift1 := "LIFT_1".Data_Current;
   "RUN_TIME_PARAM".Current_Lift2 := "LIFT_2".Data_Current;
   "RUN_TIME_PARAM".Current_Lift3 := "LIFT_3".Data_Current;
END_REGION

REGION Network 11: TRANFER 2
   RUNG wire#powerrail
      Contact( "Axis_X".All_Done )
      Contact( "Tranfer_1".All_Done )
      Contact( "Axis_Lift".All_Done )
      Contact( "LIFT_1".All_Done )
      Contact( "LIFT_2".All_Done )
      Contact( "LIFT_3".All_Done )
      "Tranfer_2"(Busy := "MB_Comunicate".Busy, Done := "MB_Comunicate".Done, Error := "MB_Comunicate".Error, Status := "MB_Comunicate".Status, Enable_block := "AlwaysTRUE", Ptr := "MB_Comunicate".DataPtr, Req => "MB_Comunicate".Req, Mb_ID => "MB_Comunicate".MB_ID, DataLen => "MB_Comunicate".DataLen, DataAddr => "MB_Comunicate".DataAddr, Mode => "MB_Comunicate".Mode)
   END_RUNG
   // the same network as SCL:
   IF "Axis_X".All_Done AND "Tranfer_1".All_Done AND "Axis_Lift".All_Done AND "LIFT_1".All_Done AND "LIFT_2".All_Done AND "LIFT_3".All_Done THEN
       "Tranfer_2"(Busy := "MB_Comunicate".Busy,   // "Inventer_Control"
                   Done := "MB_Comunicate".Done,
                   Error := "MB_Comunicate".Error,
                   Status := "MB_Comunicate".Status,
                   Enable_block := "AlwaysTRUE",
                   Ptr := "MB_Comunicate".DataPtr,
                   Req => "MB_Comunicate".Req,
                   Mb_ID => "MB_Comunicate".MB_ID,
                   DataLen => "MB_Comunicate".DataLen,
                   DataAddr => "MB_Comunicate".DataAddr,
                   Mode => "MB_Comunicate".Mode);
   END_IF;
END_REGION

REGION Network 12: Axis X Home
   RUNG wire#powerrail
      Contact( "MANUAL_STATE" )
      Contact( "HOME_MAN_TRIGGER_PC" )
      wire#w1
      { S7_Templates := "SrcType := Int" } EQ_Contact(in1 := "SELECT_AXIS_HOME", in2 := 0)
      wire#w2
      Contact( "SS Up XL Robot" )
      P_Trig( "Edge_2" )
      wire#w3
      S_Coil( "Axis_X".Move_Home )
   END_RUNG
   RUNG wire#w1
      { S7_Templates := "SrcType := Int" } EQ_Contact(in1 := "SELECT_AXIS_HOME", in2 := 1)
   END_RUNG wire#w2
   RUNG wire#powerrail
      Contact( "AUTO_STATE" )
      Contact( "HOME_AUTO_TRIGGER_PC" )
   END_RUNG wire#w2
   RUNG wire#w3
      R_Coil( "HOME_MAN_TRIGGER_PC" )
   END_RUNG
   // the same network as SCL:
   #_w1 := (("MANUAL_STATE" AND "HOME_MAN_TRIGGER_PC" AND (("SELECT_AXIS_HOME" = 0) OR ("SELECT_AXIS_HOME" = 1))) OR ("AUTO_STATE" AND "HOME_AUTO_TRIGGER_PC")) AND "SS Up XL Robot";
   #_w2 := #_w1 AND NOT "Edge_2";   // rising edge
   "Edge_2" := #_w1;
   IF #_w2 THEN
       "Axis_X".Move_Home := TRUE;
       "HOME_MAN_TRIGGER_PC" := FALSE;
   END_IF;
END_REGION

REGION Network 13: AXIS LIFT HOME
   RUNG wire#powerrail
      Contact( "MANUAL_STATE" )
      Contact( "HOME_MAN_TRIGGER_PC" )
      wire#w1
      { S7_Templates := "SrcType := Int" } EQ_Contact(in1 := "SELECT_AXIS_HOME", in2 := 0)
      wire#w2
      P_Trig( "Edge_2" )
      wire#w3
      S_Coil( "Axis_Lift".Move_Home )
   END_RUNG
   RUNG wire#w1
      { S7_Templates := "SrcType := Int" } EQ_Contact(in1 := "SELECT_AXIS_HOME", in2 := 2)
   END_RUNG wire#w2
   RUNG wire#powerrail
      Contact( "AUTO_STATE" )
      Contact( "HOME_AUTO_TRIGGER_PC" )
   END_RUNG wire#w2
   RUNG wire#w3
      R_Coil( "HOME_MAN_TRIGGER_PC" )
   END_RUNG
   // the same network as SCL:
   #_w1 := ("MANUAL_STATE" AND "HOME_MAN_TRIGGER_PC" AND (("SELECT_AXIS_HOME" = 0) OR ("SELECT_AXIS_HOME" = 2))) OR ("AUTO_STATE" AND "HOME_AUTO_TRIGGER_PC");
   #_w2 := #_w1 AND NOT "Edge_2";   // rising edge
   "Edge_2" := #_w1;
   IF #_w2 THEN
       "Axis_Lift".Move_Home := TRUE;
       "HOME_MAN_TRIGGER_PC" := FALSE;
   END_IF;
END_REGION

REGION Network 14: JOG X VS LIFT
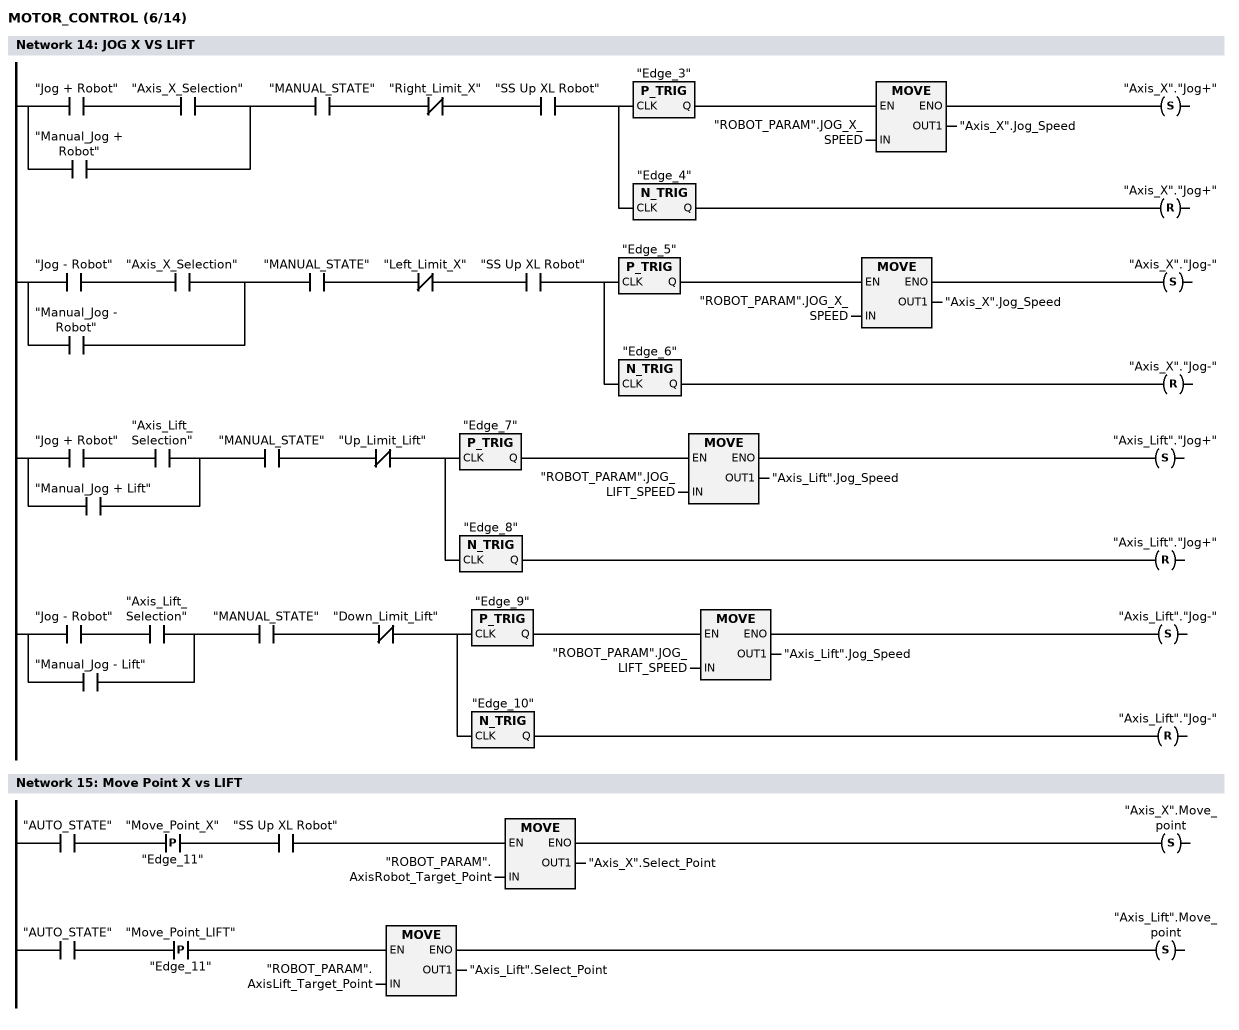
   RUNG wire#powerrail
      Contact( "Jog + Robot" )
      Contact( "Axis_X_Selection" )
      wire#w1
      Contact( "MANUAL_STATE" )
      I_Contact( "Right_Limit_X" )
      Contact( "SS Up XL Robot" )
      wire#w2
      P_Trig( "Edge_3" )
      { S7_GenerateENO := "TRUE" } Move(in := "ROBOT_PARAM".JOG_X_SPEED, out1 => "Axis_X".Jog_Speed)
      S_Coil( "Axis_X"."Jog+" )
   END_RUNG
   RUNG wire#powerrail
      Contact( "Manual_Jog + Robot" )
   END_RUNG wire#w1
   RUNG wire#w2
      N_Trig( "Edge_4" )
      R_Coil( "Axis_X"."Jog+" )
   END_RUNG
   RUNG wire#powerrail
      Contact( "Jog - Robot" )
      Contact( "Axis_X_Selection" )
      wire#w3
      Contact( "MANUAL_STATE" )
      I_Contact( "Left_Limit_X" )
      Contact( "SS Up XL Robot" )
      wire#w4
      P_Trig( "Edge_5" )
      { S7_GenerateENO := "TRUE" } Move(in := "ROBOT_PARAM".JOG_X_SPEED, out1 => "Axis_X".Jog_Speed)
      S_Coil( "Axis_X"."Jog-" )
   END_RUNG
   RUNG wire#powerrail
      Contact( "Manual_Jog - Robot" )
   END_RUNG wire#w3
   RUNG wire#w4
      N_Trig( "Edge_6" )
      R_Coil( "Axis_X"."Jog-" )
   END_RUNG
   RUNG wire#powerrail
      Contact( "Jog + Robot" )
      Contact( "Axis_Lift_Selection" )
      wire#w5
      Contact( "MANUAL_STATE" )
      I_Contact( "Up_Limit_Lift" )
      wire#w6
      P_Trig( "Edge_7" )
      { S7_GenerateENO := "TRUE" } Move(in := "ROBOT_PARAM".JOG_LIFT_SPEED, out1 => "Axis_Lift".Jog_Speed)
      S_Coil( "Axis_Lift"."Jog+" )
   END_RUNG
   RUNG wire#powerrail
      Contact( "Manual_Jog + Lift" )
   END_RUNG wire#w5
   RUNG wire#w6
      N_Trig( "Edge_8" )
      R_Coil( "Axis_Lift"."Jog+" )
   END_RUNG
   RUNG wire#powerrail
      Contact( "Jog - Robot" )
      Contact( "Axis_Lift_Selection" )
      wire#w7
      Contact( "MANUAL_STATE" )
      I_Contact( "Down_Limit_Lift" )
      wire#w8
      P_Trig( "Edge_9" )
      { S7_GenerateENO := "TRUE" } Move(in := "ROBOT_PARAM".JOG_LIFT_SPEED, out1 => "Axis_Lift".Jog_Speed)
      S_Coil( "Axis_Lift"."Jog-" )
   END_RUNG
   RUNG wire#powerrail
      Contact( "Manual_Jog - Lift" )
   END_RUNG wire#w7
   RUNG wire#w8
      N_Trig( "Edge_10" )
      R_Coil( "Axis_Lift"."Jog-" )
   END_RUNG
   // the same network as SCL:
   // ENO of a box is taken as its EN; it also drops when the box reports an error
   #_w1 := (("Jog + Robot" AND "Axis_X_Selection") OR "Manual_Jog + Robot") AND "MANUAL_STATE" AND NOT "Right_Limit_X" AND "SS Up XL Robot";
   #_w2 := #_w1 AND NOT "Edge_3";   // rising edge
   "Edge_3" := #_w1;
   IF #_w2 THEN
       "Axis_X".Jog_Speed := "ROBOT_PARAM".JOG_X_SPEED;
       "Axis_X"."Jog+" := TRUE;
   END_IF;
   #_w3 := NOT #_w1 AND "Edge_4";   // falling edge
   "Edge_4" := #_w1;
   IF #_w3 THEN "Axis_X"."Jog+" := FALSE; END_IF;
   #_w4 := (("Jog - Robot" AND "Axis_X_Selection") OR "Manual_Jog - Robot") AND "MANUAL_STATE" AND NOT "Left_Limit_X" AND "SS Up XL Robot";
   #_w5 := #_w4 AND NOT "Edge_5";   // rising edge
   "Edge_5" := #_w4;
   IF #_w5 THEN
       "Axis_X".Jog_Speed := "ROBOT_PARAM".JOG_X_SPEED;
       "Axis_X"."Jog-" := TRUE;
   END_IF;
   #_w6 := NOT #_w4 AND "Edge_6";   // falling edge
   "Edge_6" := #_w4;
   IF #_w6 THEN "Axis_X"."Jog-" := FALSE; END_IF;
   #_w7 := (("Jog + Robot" AND "Axis_Lift_Selection") OR "Manual_Jog + Lift") AND "MANUAL_STATE" AND NOT "Up_Limit_Lift";
   #_w8 := #_w7 AND NOT "Edge_7";   // rising edge
   "Edge_7" := #_w7;
   IF #_w8 THEN
       "Axis_Lift".Jog_Speed := "ROBOT_PARAM".JOG_LIFT_SPEED;
       "Axis_Lift"."Jog+" := TRUE;
   END_IF;
   #_w9 := NOT #_w7 AND "Edge_8";   // falling edge
   "Edge_8" := #_w7;
   IF #_w9 THEN "Axis_Lift"."Jog+" := FALSE; END_IF;
   #_w10 := (("Jog - Robot" AND "Axis_Lift_Selection") OR "Manual_Jog - Lift") AND "MANUAL_STATE" AND NOT "Down_Limit_Lift";
   #_w11 := #_w10 AND NOT "Edge_9";   // rising edge
   "Edge_9" := #_w10;
   IF #_w11 THEN
       "Axis_Lift".Jog_Speed := "ROBOT_PARAM".JOG_LIFT_SPEED;
       "Axis_Lift"."Jog-" := TRUE;
   END_IF;
   #_w12 := NOT #_w10 AND "Edge_10";   // falling edge
   "Edge_10" := #_w10;
   IF #_w12 THEN "Axis_Lift"."Jog-" := FALSE; END_IF;
END_REGION

REGION Network 15: Move Point X vs LIFT
   RUNG wire#powerrail
      Contact( "AUTO_STATE" )
      P_Contact(operand := "Move_Point_X", bit := "Edge_11")
      Contact( "SS Up XL Robot" )
      { S7_GenerateENO := "TRUE" } Move(in := "ROBOT_PARAM".AxisRobot_Target_Point, out1 => "Axis_X".Select_Point)
      S_Coil( "Axis_X".Move_point )
   END_RUNG
   RUNG wire#powerrail
      Contact( "AUTO_STATE" )
      P_Contact(operand := "Move_Point_LIFT", bit := "Edge_11")
      { S7_GenerateENO := "TRUE" } Move(in := "ROBOT_PARAM".AxisLift_Target_Point, out1 => "Axis_Lift".Select_Point)
      S_Coil( "Axis_Lift".Move_point )
   END_RUNG
   // the same network as SCL:
   // ENO of a box is taken as its EN; it also drops when the box reports an error
   #_w1 := "AUTO_STATE" AND "Move_Point_X" AND NOT "Edge_11";   // rising edge of "Move_Point_X"
   "Edge_11" := "Move_Point_X";
   IF #_w1 AND "SS Up XL Robot" THEN
       "Axis_X".Select_Point := "ROBOT_PARAM".AxisRobot_Target_Point;
       "Axis_X".Move_point := TRUE;
   END_IF;
   #_w2 := "AUTO_STATE" AND "Move_Point_LIFT" AND NOT "Edge_11";   // rising edge of "Move_Point_LIFT"
   "Edge_11" := "Move_Point_LIFT";
   IF #_w2 THEN
       "Axis_Lift".Select_Point := "ROBOT_PARAM".AxisLift_Target_Point;
       "Axis_Lift".Move_point := TRUE;
   END_IF;
END_REGION

REGION Network 16: SetPoint X vs LIFT
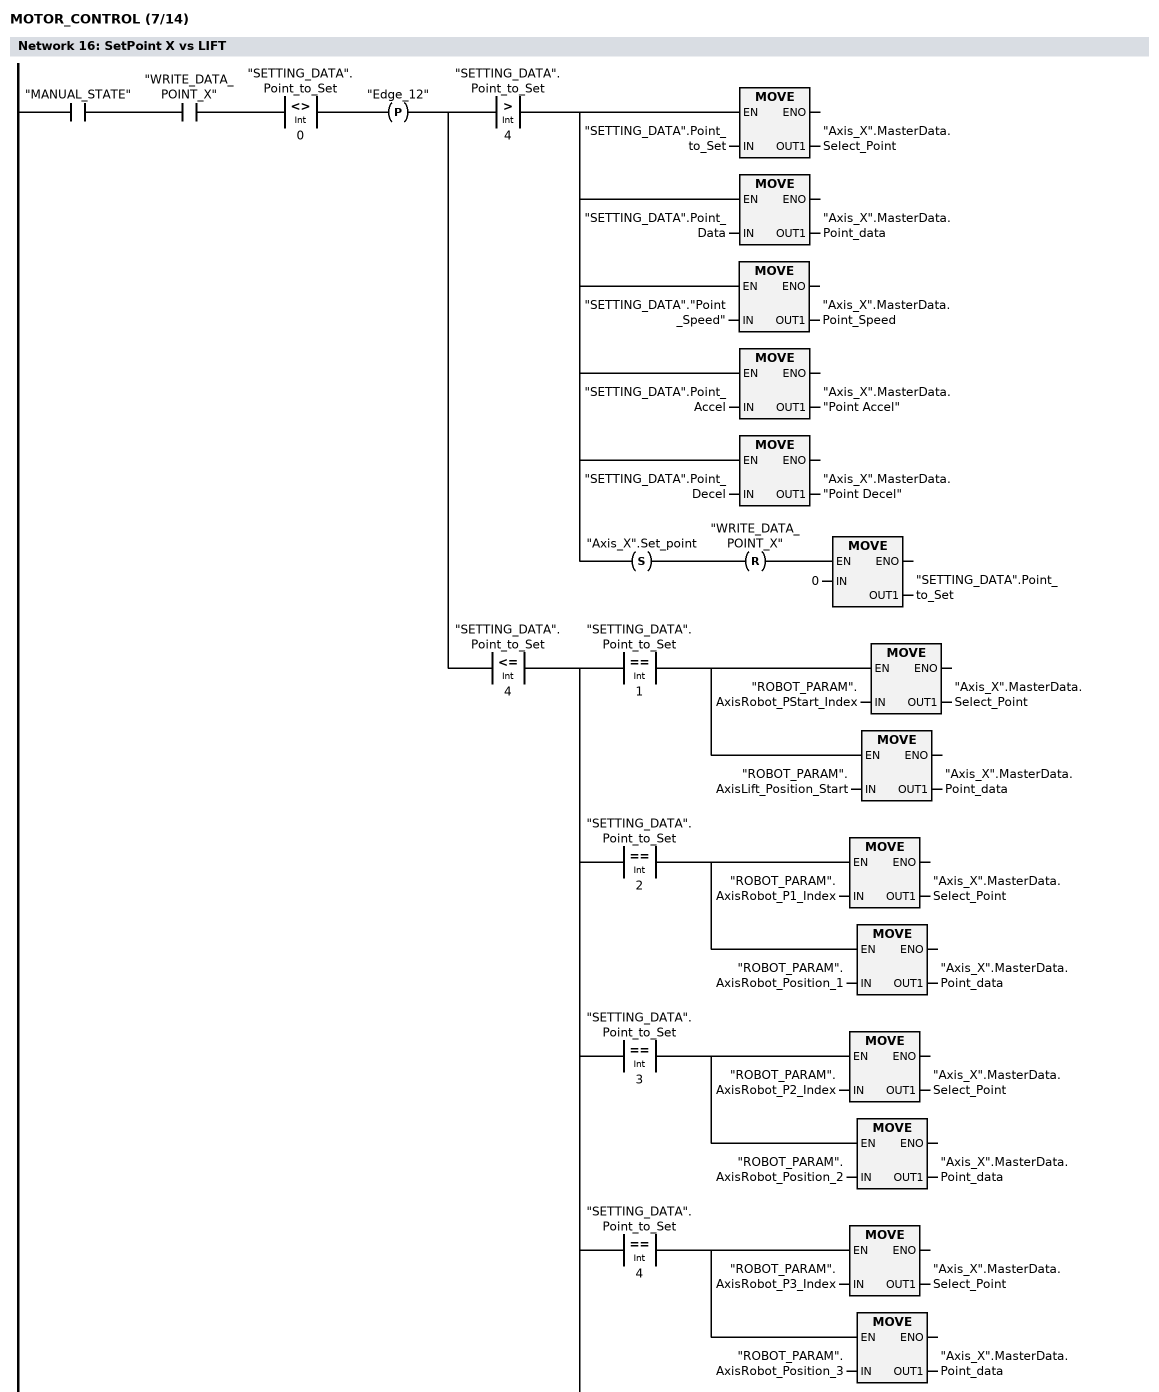
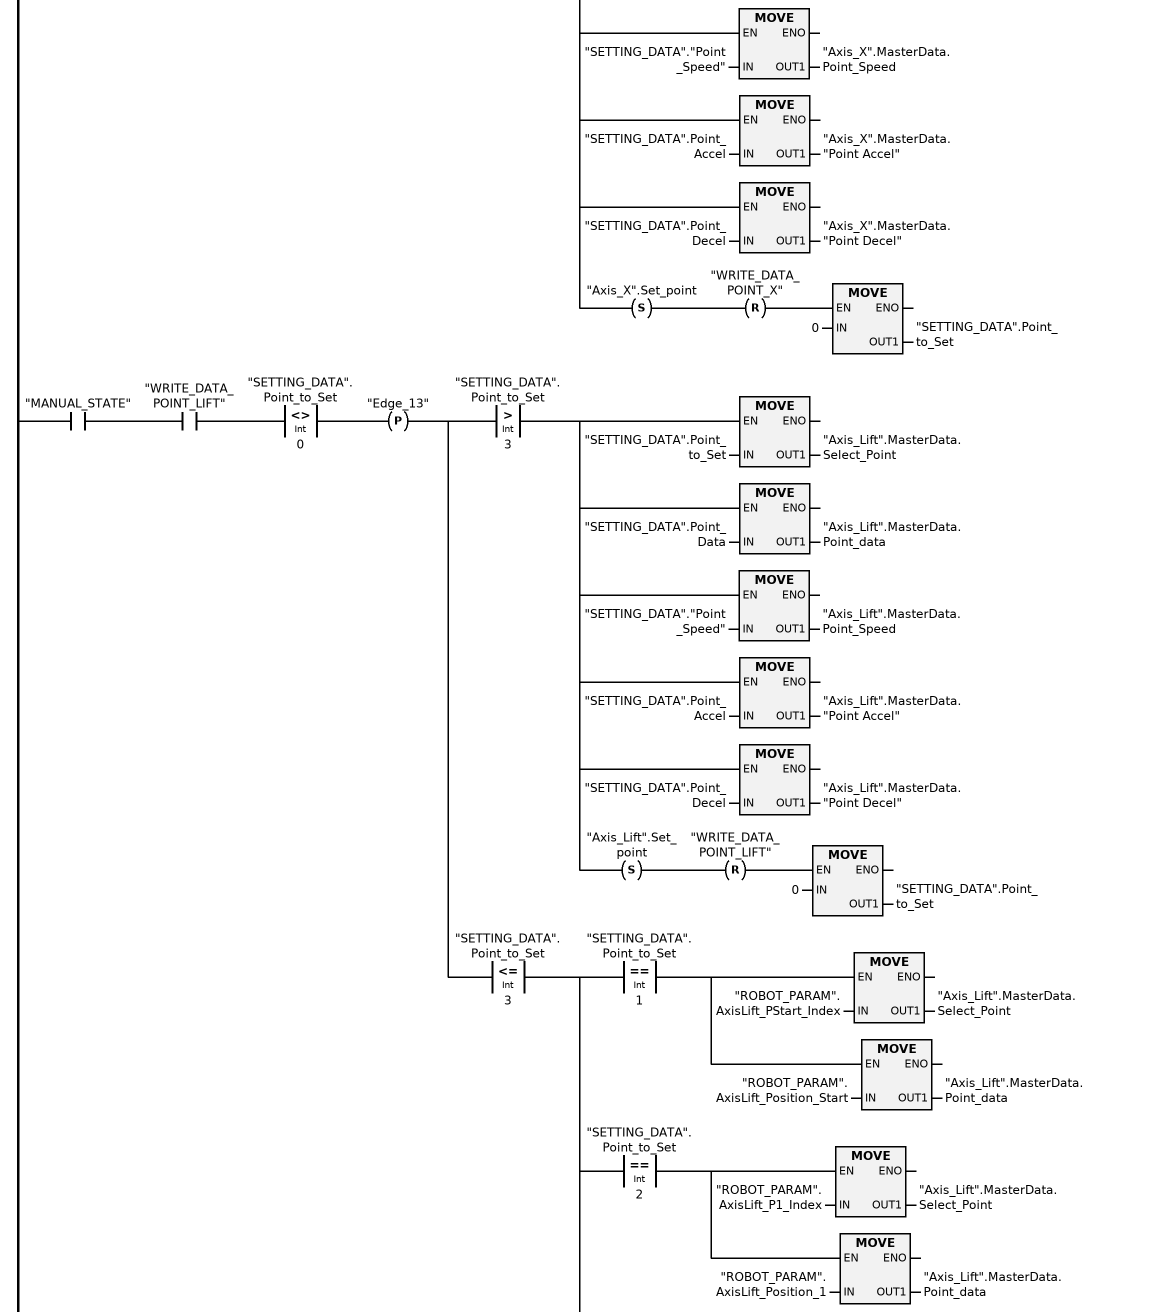
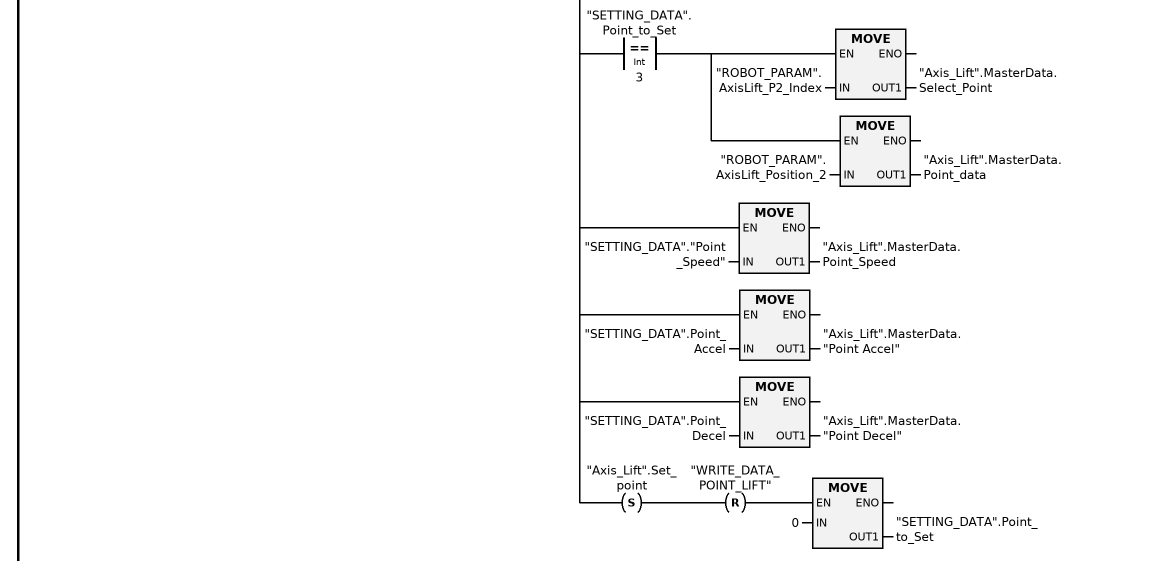
   RUNG wire#powerrail
      Contact( "MANUAL_STATE" )
      Contact( "WRITE_DATA_POINT_X" )
      { S7_Templates := "SrcType := Int" } NE_Contact(in1 := "SETTING_DATA".Point_to_Set, in2 := 0)
      P_Trig( "Edge_12" )
      wire#w1
      { S7_Templates := "SrcType := Int" } GT_Contact(in1 := "SETTING_DATA".Point_to_Set, in2 := 4)
      wire#w2
      { S7_GenerateENO := "TRUE" } Move(in := "SETTING_DATA".Point_to_Set, out1 => "Axis_X".MasterData.Select_Point)
   END_RUNG
   RUNG wire#w2
      { S7_GenerateENO := "TRUE" } Move(in := "SETTING_DATA".Point_Data, out1 => "Axis_X".MasterData.Point_data)
   END_RUNG
   RUNG wire#w2
      { S7_GenerateENO := "TRUE" } Move(in := "SETTING_DATA"."Point _Speed", out1 => "Axis_X".MasterData.Point_Speed)
   END_RUNG
   RUNG wire#w2
      { S7_GenerateENO := "TRUE" } Move(in := "SETTING_DATA".Point_Accel, out1 => "Axis_X".MasterData."Point Accel")
   END_RUNG
   RUNG wire#w2
      { S7_GenerateENO := "TRUE" } Move(in := "SETTING_DATA".Point_Decel, out1 => "Axis_X".MasterData."Point Decel")
   END_RUNG
   RUNG wire#w2
      S_Coil( "Axis_X".Set_point )
      R_Coil( "WRITE_DATA_POINT_X" )
      { S7_GenerateENO := "TRUE" } Move(in := 0, out1 => "SETTING_DATA".Point_to_Set)
   END_RUNG
   RUNG wire#w1
      { S7_Templates := "SrcType := Int" } LE_Contact(in1 := "SETTING_DATA".Point_to_Set, in2 := 4)
      wire#w3
      { S7_Templates := "SrcType := Int" } EQ_Contact(in1 := "SETTING_DATA".Point_to_Set, in2 := 1)
      wire#w4
      { S7_GenerateENO := "TRUE" } Move(in := "ROBOT_PARAM".AxisRobot_PStart_Index, out1 => "Axis_X".MasterData.Select_Point)
   END_RUNG
   RUNG wire#w4
      { S7_GenerateENO := "TRUE" } Move(in := "ROBOT_PARAM".AxisLift_Position_Start, out1 => "Axis_X".MasterData.Point_data)
   END_RUNG
   RUNG wire#w3
      { S7_Templates := "SrcType := Int" } EQ_Contact(in1 := "SETTING_DATA".Point_to_Set, in2 := 2)
      wire#w5
      { S7_GenerateENO := "TRUE" } Move(in := "ROBOT_PARAM".AxisRobot_P1_Index, out1 => "Axis_X".MasterData.Select_Point)
   END_RUNG
   RUNG wire#w5
      { S7_GenerateENO := "TRUE" } Move(in := "ROBOT_PARAM".AxisRobot_Position_1, out1 => "Axis_X".MasterData.Point_data)
   END_RUNG
   RUNG wire#w3
      { S7_Templates := "SrcType := Int" } EQ_Contact(in1 := "SETTING_DATA".Point_to_Set, in2 := 3)
      wire#w6
      { S7_GenerateENO := "TRUE" } Move(in := "ROBOT_PARAM".AxisRobot_P2_Index, out1 => "Axis_X".MasterData.Select_Point)
   END_RUNG
   RUNG wire#w6
      { S7_GenerateENO := "TRUE" } Move(in := "ROBOT_PARAM".AxisRobot_Position_2, out1 => "Axis_X".MasterData.Point_data)
   END_RUNG
   RUNG wire#w3
      { S7_Templates := "SrcType := Int" } EQ_Contact(in1 := "SETTING_DATA".Point_to_Set, in2 := 4)
      wire#w7
      { S7_GenerateENO := "TRUE" } Move(in := "ROBOT_PARAM".AxisRobot_P3_Index, out1 => "Axis_X".MasterData.Select_Point)
   END_RUNG
   RUNG wire#w7
      { S7_GenerateENO := "TRUE" } Move(in := "ROBOT_PARAM".AxisRobot_Position_3, out1 => "Axis_X".MasterData.Point_data)
   END_RUNG
   RUNG wire#w3
      { S7_GenerateENO := "TRUE" } Move(in := "SETTING_DATA"."Point _Speed", out1 => "Axis_X".MasterData.Point_Speed)
   END_RUNG
   RUNG wire#w3
      { S7_GenerateENO := "TRUE" } Move(in := "SETTING_DATA".Point_Accel, out1 => "Axis_X".MasterData."Point Accel")
   END_RUNG
   RUNG wire#w3
      { S7_GenerateENO := "TRUE" } Move(in := "SETTING_DATA".Point_Decel, out1 => "Axis_X".MasterData."Point Decel")
   END_RUNG
   RUNG wire#w3
      S_Coil( "Axis_X".Set_point )
      R_Coil( "WRITE_DATA_POINT_X" )
      { S7_GenerateENO := "TRUE" } Move(in := 0, out1 => "SETTING_DATA".Point_to_Set)
   END_RUNG
   RUNG wire#powerrail
      Contact( "MANUAL_STATE" )
      Contact( "WRITE_DATA_POINT_LIFT" )
      { S7_Templates := "SrcType := Int" } NE_Contact(in1 := "SETTING_DATA".Point_to_Set, in2 := 0)
      P_Trig( "Edge_13" )
      wire#w8
      { S7_Templates := "SrcType := Int" } GT_Contact(in1 := "SETTING_DATA".Point_to_Set, in2 := 3)
      wire#w9
      { S7_GenerateENO := "TRUE" } Move(in := "SETTING_DATA".Point_to_Set, out1 => "Axis_Lift".MasterData.Select_Point)
   END_RUNG
   RUNG wire#w9
      { S7_GenerateENO := "TRUE" } Move(in := "SETTING_DATA".Point_Data, out1 => "Axis_Lift".MasterData.Point_data)
   END_RUNG
   RUNG wire#w9
      { S7_GenerateENO := "TRUE" } Move(in := "SETTING_DATA"."Point _Speed", out1 => "Axis_Lift".MasterData.Point_Speed)
   END_RUNG
   RUNG wire#w9
      { S7_GenerateENO := "TRUE" } Move(in := "SETTING_DATA".Point_Accel, out1 => "Axis_Lift".MasterData."Point Accel")
   END_RUNG
   RUNG wire#w9
      { S7_GenerateENO := "TRUE" } Move(in := "SETTING_DATA".Point_Decel, out1 => "Axis_Lift".MasterData."Point Decel")
   END_RUNG
   RUNG wire#w9
      S_Coil( "Axis_Lift".Set_point )
      R_Coil( "WRITE_DATA_POINT_LIFT" )
      { S7_GenerateENO := "TRUE" } Move(in := 0, out1 => "SETTING_DATA".Point_to_Set)
   END_RUNG
   RUNG wire#w8
      { S7_Templates := "SrcType := Int" } LE_Contact(in1 := "SETTING_DATA".Point_to_Set, in2 := 3)
      wire#w10
      { S7_Templates := "SrcType := Int" } EQ_Contact(in1 := "SETTING_DATA".Point_to_Set, in2 := 1)
      wire#w11
      { S7_GenerateENO := "TRUE" } Move(in := "ROBOT_PARAM".AxisLift_PStart_Index, out1 => "Axis_Lift".MasterData.Select_Point)
   END_RUNG
   RUNG wire#w11
      { S7_GenerateENO := "TRUE" } Move(in := "ROBOT_PARAM".AxisLift_Position_Start, out1 => "Axis_Lift".MasterData.Point_data)
   END_RUNG
   RUNG wire#w10
      { S7_Templates := "SrcType := Int" } EQ_Contact(in1 := "SETTING_DATA".Point_to_Set, in2 := 2)
      wire#w12
      { S7_GenerateENO := "TRUE" } Move(in := "ROBOT_PARAM".AxisLift_P1_Index, out1 => "Axis_Lift".MasterData.Select_Point)
   END_RUNG
   RUNG wire#w12
      { S7_GenerateENO := "TRUE" } Move(in := "ROBOT_PARAM".AxisLift_Position_1, out1 => "Axis_Lift".MasterData.Point_data)
   END_RUNG
   RUNG wire#w10
      { S7_Templates := "SrcType := Int" } EQ_Contact(in1 := "SETTING_DATA".Point_to_Set, in2 := 3)
      wire#w13
      { S7_GenerateENO := "TRUE" } Move(in := "ROBOT_PARAM".AxisLift_P2_Index, out1 => "Axis_Lift".MasterData.Select_Point)
   END_RUNG
   RUNG wire#w13
      { S7_GenerateENO := "TRUE" } Move(in := "ROBOT_PARAM".AxisLift_Position_2, out1 => "Axis_Lift".MasterData.Point_data)
   END_RUNG
   RUNG wire#w10
      { S7_GenerateENO := "TRUE" } Move(in := "SETTING_DATA"."Point _Speed", out1 => "Axis_Lift".MasterData.Point_Speed)
   END_RUNG
   RUNG wire#w10
      { S7_GenerateENO := "TRUE" } Move(in := "SETTING_DATA".Point_Accel, out1 => "Axis_Lift".MasterData."Point Accel")
   END_RUNG
   RUNG wire#w10
      { S7_GenerateENO := "TRUE" } Move(in := "SETTING_DATA".Point_Decel, out1 => "Axis_Lift".MasterData."Point Decel")
   END_RUNG
   RUNG wire#w10
      S_Coil( "Axis_Lift".Set_point )
      R_Coil( "WRITE_DATA_POINT_LIFT" )
      { S7_GenerateENO := "TRUE" } Move(in := 0, out1 => "SETTING_DATA".Point_to_Set)
   END_RUNG
   // the same network as SCL:
   #_w1 := "MANUAL_STATE" AND "WRITE_DATA_POINT_X" AND ("SETTING_DATA".Point_to_Set <> 0);
   #_w2 := #_w1 AND NOT "Edge_12";   // rising edge
   "Edge_12" := #_w1;
   IF #_w2 AND ("SETTING_DATA".Point_to_Set > 4) THEN
       "Axis_X".MasterData.Select_Point := "SETTING_DATA".Point_to_Set;
       "Axis_X".MasterData.Point_data := "SETTING_DATA".Point_Data;
       "Axis_X".MasterData.Point_Speed := "SETTING_DATA"."Point _Speed";
       "Axis_X".MasterData."Point Accel" := "SETTING_DATA".Point_Accel;
       "Axis_X".MasterData."Point Decel" := "SETTING_DATA".Point_Decel;
       "Axis_X".Set_point := TRUE;
       "WRITE_DATA_POINT_X" := FALSE;
       "SETTING_DATA".Point_to_Set := 0;
   END_IF;
   #_w3 := #_w2 AND ("SETTING_DATA".Point_to_Set <= 4);
   IF #_w3 AND ("SETTING_DATA".Point_to_Set = 1) THEN
       "Axis_X".MasterData.Select_Point := "ROBOT_PARAM".AxisRobot_PStart_Index;
       "Axis_X".MasterData.Point_data := "ROBOT_PARAM".AxisLift_Position_Start;
   END_IF;
   IF #_w3 AND ("SETTING_DATA".Point_to_Set = 2) THEN
       "Axis_X".MasterData.Select_Point := "ROBOT_PARAM".AxisRobot_P1_Index;
       "Axis_X".MasterData.Point_data := "ROBOT_PARAM".AxisRobot_Position_1;
   END_IF;
   IF #_w3 AND ("SETTING_DATA".Point_to_Set = 3) THEN
       "Axis_X".MasterData.Select_Point := "ROBOT_PARAM".AxisRobot_P2_Index;
       "Axis_X".MasterData.Point_data := "ROBOT_PARAM".AxisRobot_Position_2;
   END_IF;
   IF #_w3 AND ("SETTING_DATA".Point_to_Set = 4) THEN
       "Axis_X".MasterData.Select_Point := "ROBOT_PARAM".AxisRobot_P3_Index;
       "Axis_X".MasterData.Point_data := "ROBOT_PARAM".AxisRobot_Position_3;
   END_IF;
   IF #_w3 THEN
       "Axis_X".MasterData.Point_Speed := "SETTING_DATA"."Point _Speed";
       "Axis_X".MasterData."Point Accel" := "SETTING_DATA".Point_Accel;
       "Axis_X".MasterData."Point Decel" := "SETTING_DATA".Point_Decel;
       "Axis_X".Set_point := TRUE;
       "WRITE_DATA_POINT_X" := FALSE;
       "SETTING_DATA".Point_to_Set := 0;
   END_IF;
   #_w4 := "MANUAL_STATE" AND "WRITE_DATA_POINT_LIFT" AND ("SETTING_DATA".Point_to_Set <> 0);
   #_w5 := #_w4 AND NOT "Edge_13";   // rising edge
   "Edge_13" := #_w4;
   IF #_w5 AND ("SETTING_DATA".Point_to_Set > 3) THEN
       "Axis_Lift".MasterData.Select_Point := "SETTING_DATA".Point_to_Set;
       "Axis_Lift".MasterData.Point_data := "SETTING_DATA".Point_Data;
       "Axis_Lift".MasterData.Point_Speed := "SETTING_DATA"."Point _Speed";
       "Axis_Lift".MasterData."Point Accel" := "SETTING_DATA".Point_Accel;
       "Axis_Lift".MasterData."Point Decel" := "SETTING_DATA".Point_Decel;
       "Axis_Lift".Set_point := TRUE;
       "WRITE_DATA_POINT_LIFT" := FALSE;
       "SETTING_DATA".Point_to_Set := 0;
   END_IF;
   #_w6 := #_w5 AND ("SETTING_DATA".Point_to_Set <= 3);
   IF #_w6 AND ("SETTING_DATA".Point_to_Set = 1) THEN
       "Axis_Lift".MasterData.Select_Point := "ROBOT_PARAM".AxisLift_PStart_Index;
       "Axis_Lift".MasterData.Point_data := "ROBOT_PARAM".AxisLift_Position_Start;
   END_IF;
   IF #_w6 AND ("SETTING_DATA".Point_to_Set = 2) THEN
       "Axis_Lift".MasterData.Select_Point := "ROBOT_PARAM".AxisLift_P1_Index;
       "Axis_Lift".MasterData.Point_data := "ROBOT_PARAM".AxisLift_Position_1;
   END_IF;
   IF #_w6 AND ("SETTING_DATA".Point_to_Set = 3) THEN
       "Axis_Lift".MasterData.Select_Point := "ROBOT_PARAM".AxisLift_P2_Index;
       "Axis_Lift".MasterData.Point_data := "ROBOT_PARAM".AxisLift_Position_2;
   END_IF;
   IF #_w6 THEN
       "Axis_Lift".MasterData.Point_Speed := "SETTING_DATA"."Point _Speed";
       "Axis_Lift".MasterData."Point Accel" := "SETTING_DATA".Point_Accel;
       "Axis_Lift".MasterData."Point Decel" := "SETTING_DATA".Point_Decel;
       "Axis_Lift".Set_point := TRUE;
       "WRITE_DATA_POINT_LIFT" := FALSE;
       "SETTING_DATA".Point_to_Set := 0;
   END_IF;
END_REGION

REGION Network 17: Start Config
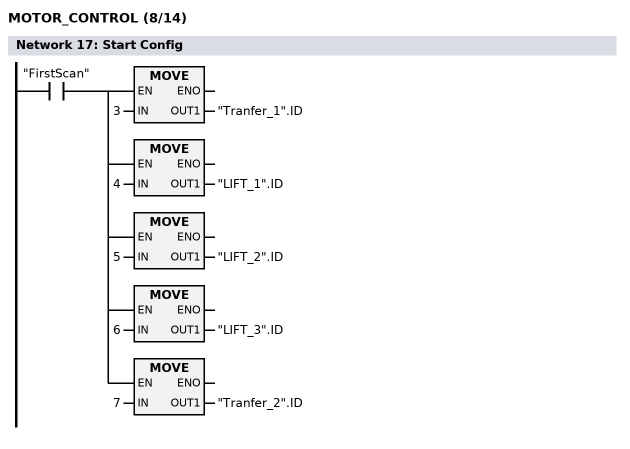
   RUNG wire#powerrail
      Contact( "FirstScan" )
      wire#w1
      { S7_GenerateENO := "TRUE" } Move(in := 3, out1 => "Tranfer_1".ID)
   END_RUNG
   RUNG wire#w1
      { S7_GenerateENO := "TRUE" } Move(in := 4, out1 => "LIFT_1".ID)
   END_RUNG
   RUNG wire#w1
      { S7_GenerateENO := "TRUE" } Move(in := 5, out1 => "LIFT_2".ID)
   END_RUNG
   RUNG wire#w1
      { S7_GenerateENO := "TRUE" } Move(in := 6, out1 => "LIFT_3".ID)
   END_RUNG
   RUNG wire#w1
      { S7_GenerateENO := "TRUE" } Move(in := 7, out1 => "Tranfer_2".ID)
   END_RUNG
   // the same network as SCL:
   IF "FirstScan" THEN
       "Tranfer_1".ID := 3;
       "LIFT_1".ID := 4;
       "LIFT_2".ID := 5;
       "LIFT_3".ID := 6;
       "Tranfer_2".ID := 7;
   END_IF;
END_REGION

REGION Network 18: Tranfer 1 vs 2 Jog/Run
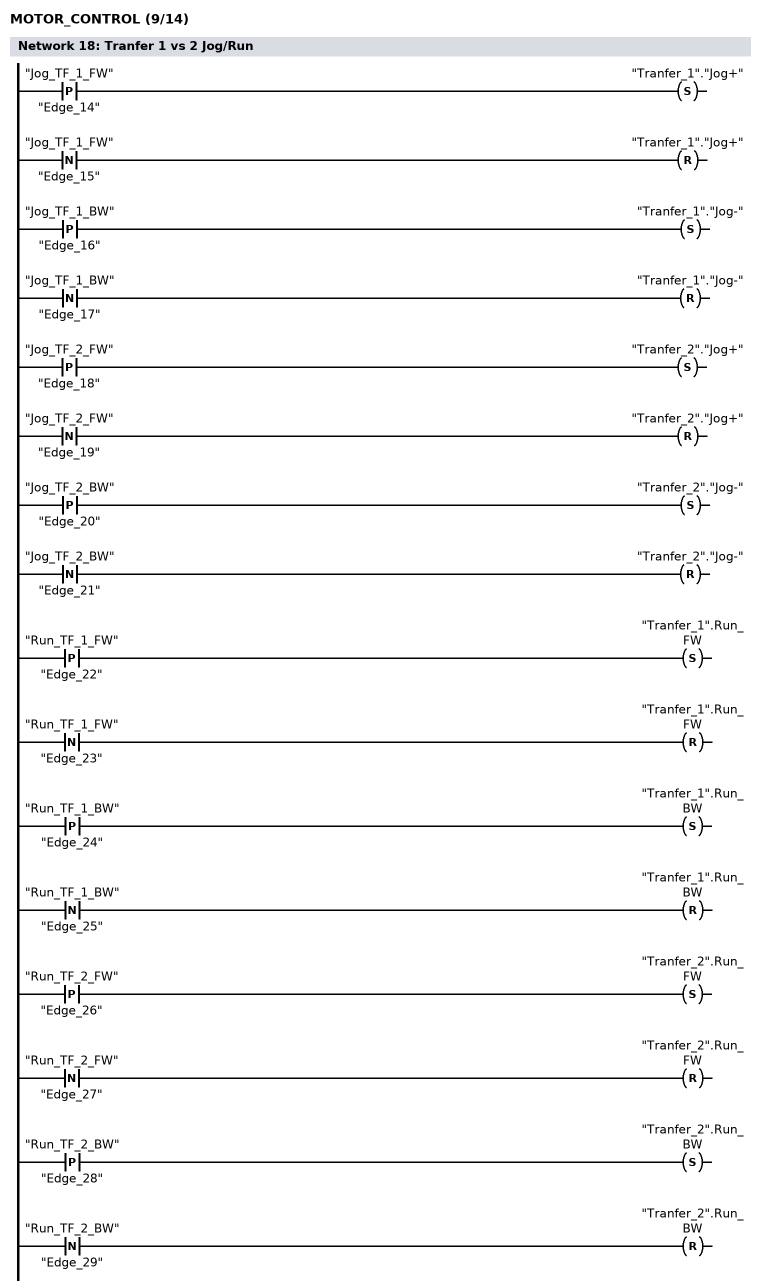
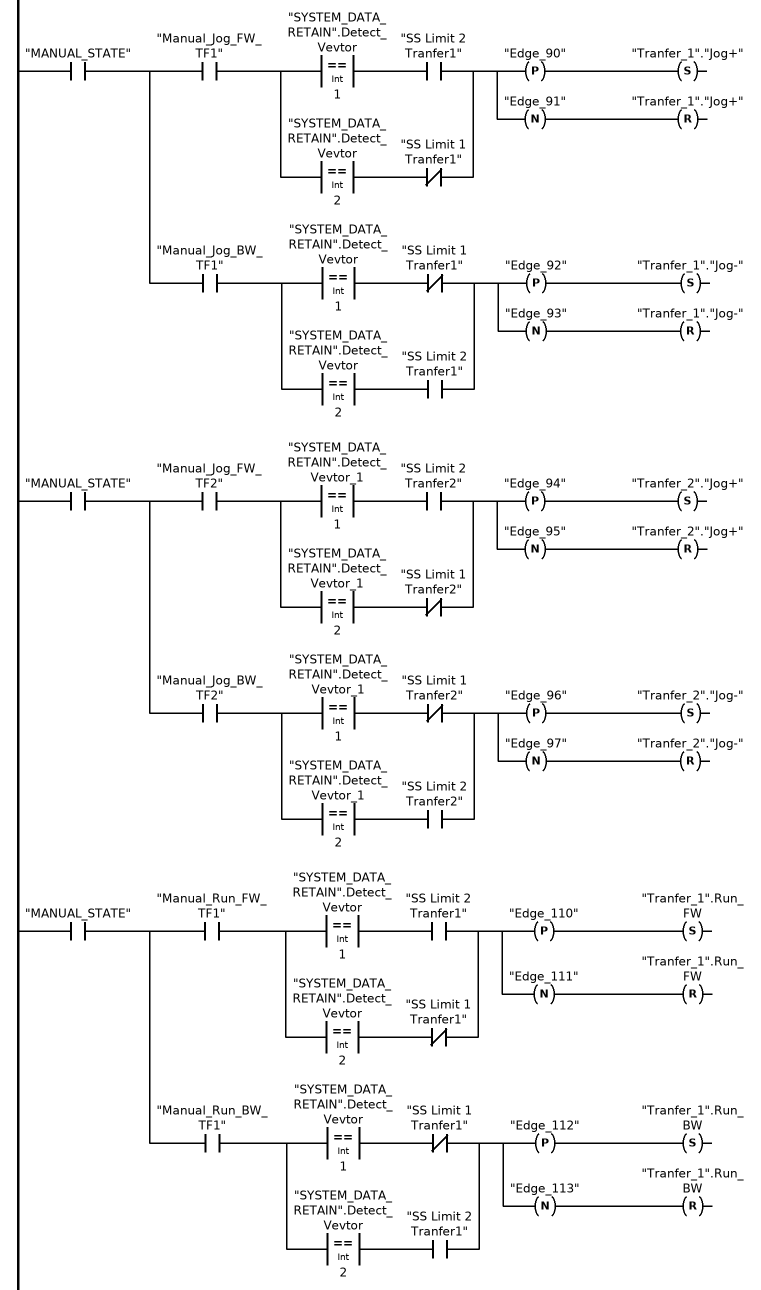
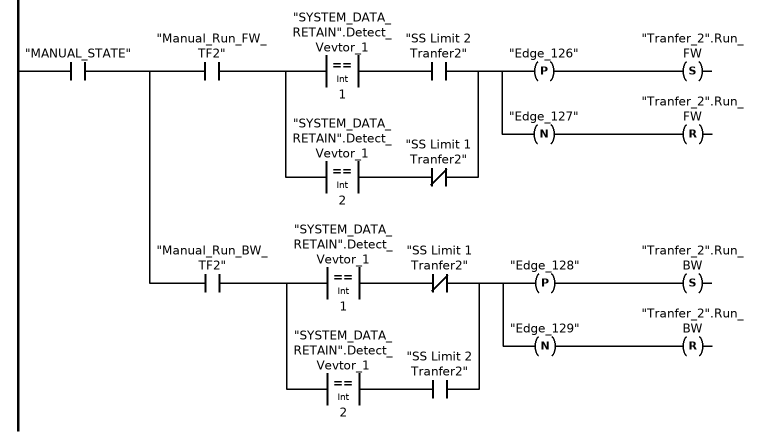
   RUNG wire#powerrail
      P_Contact(operand := "Jog_TF_1_FW", bit := "Edge_14")
      S_Coil( "Tranfer_1"."Jog+" )
   END_RUNG
   RUNG wire#powerrail
      N_Contact(operand := "Jog_TF_1_FW", bit := "Edge_15")
      R_Coil( "Tranfer_1"."Jog+" )
   END_RUNG
   RUNG wire#powerrail
      P_Contact(operand := "Jog_TF_1_BW", bit := "Edge_16")
      S_Coil( "Tranfer_1"."Jog-" )
   END_RUNG
   RUNG wire#powerrail
      N_Contact(operand := "Jog_TF_1_BW", bit := "Edge_17")
      R_Coil( "Tranfer_1"."Jog-" )
   END_RUNG
   RUNG wire#powerrail
      P_Contact(operand := "Jog_TF_2_FW", bit := "Edge_18")
      S_Coil( "Tranfer_2"."Jog+" )
   END_RUNG
   RUNG wire#powerrail
      N_Contact(operand := "Jog_TF_2_FW", bit := "Edge_19")
      R_Coil( "Tranfer_2"."Jog+" )
   END_RUNG
   RUNG wire#powerrail
      P_Contact(operand := "Jog_TF_2_BW", bit := "Edge_20")
      S_Coil( "Tranfer_2"."Jog-" )
   END_RUNG
   RUNG wire#powerrail
      N_Contact(operand := "Jog_TF_2_BW", bit := "Edge_21")
      R_Coil( "Tranfer_2"."Jog-" )
   END_RUNG
   RUNG wire#powerrail
      P_Contact(operand := "Run_TF_1_FW", bit := "Edge_22")
      S_Coil( "Tranfer_1".Run_FW )
   END_RUNG
   RUNG wire#powerrail
      N_Contact(operand := "Run_TF_1_FW", bit := "Edge_23")
      R_Coil( "Tranfer_1".Run_FW )
   END_RUNG
   RUNG wire#powerrail
      P_Contact(operand := "Run_TF_1_BW", bit := "Edge_24")
      S_Coil( "Tranfer_1".Run_BW )
   END_RUNG
   RUNG wire#powerrail
      N_Contact(operand := "Run_TF_1_BW", bit := "Edge_25")
      R_Coil( "Tranfer_1".Run_BW )
   END_RUNG
   RUNG wire#powerrail
      P_Contact(operand := "Run_TF_2_FW", bit := "Edge_26")
      S_Coil( "Tranfer_2".Run_FW )
   END_RUNG
   RUNG wire#powerrail
      N_Contact(operand := "Run_TF_2_FW", bit := "Edge_27")
      R_Coil( "Tranfer_2".Run_FW )
   END_RUNG
   RUNG wire#powerrail
      P_Contact(operand := "Run_TF_2_BW", bit := "Edge_28")
      S_Coil( "Tranfer_2".Run_BW )
   END_RUNG
   RUNG wire#powerrail
      N_Contact(operand := "Run_TF_2_BW", bit := "Edge_29")
      R_Coil( "Tranfer_2".Run_BW )
   END_RUNG
   RUNG wire#powerrail
      Contact( "MANUAL_STATE" )
      wire#w1
      Contact( "Manual_Jog_FW_TF1" )
      wire#w2
      { S7_Templates := "SrcType := Int" } EQ_Contact(in1 := "SYSTEM_DATA_RETAIN".Detect_Vevtor, in2 := 1)
      Contact( "SS Limit 2 Tranfer1" )
      wire#w3
      P_Trig( "Edge_90" )
      S_Coil( "Tranfer_1"."Jog+" )
   END_RUNG
   RUNG wire#w2
      { S7_Templates := "SrcType := Int" } EQ_Contact(in1 := "SYSTEM_DATA_RETAIN".Detect_Vevtor, in2 := 2)
      I_Contact( "SS Limit 1 Tranfer1" )
   END_RUNG wire#w3
   RUNG wire#w3
      N_Trig( "Edge_91" )
      R_Coil( "Tranfer_1"."Jog+" )
   END_RUNG
   RUNG wire#w1
      Contact( "Manual_Jog_BW_TF1" )
      wire#w4
      { S7_Templates := "SrcType := Int" } EQ_Contact(in1 := "SYSTEM_DATA_RETAIN".Detect_Vevtor, in2 := 1)
      I_Contact( "SS Limit 1 Tranfer1" )
      wire#w5
      P_Trig( "Edge_92" )
      S_Coil( "Tranfer_1"."Jog-" )
   END_RUNG
   RUNG wire#w4
      { S7_Templates := "SrcType := Int" } EQ_Contact(in1 := "SYSTEM_DATA_RETAIN".Detect_Vevtor, in2 := 2)
      Contact( "SS Limit 2 Tranfer1" )
   END_RUNG wire#w5
   RUNG wire#w5
      N_Trig( "Edge_93" )
      R_Coil( "Tranfer_1"."Jog-" )
   END_RUNG
   RUNG wire#powerrail
      Contact( "MANUAL_STATE" )
      wire#w6
      Contact( "Manual_Jog_FW_TF2" )
      wire#w7
      { S7_Templates := "SrcType := Int" } EQ_Contact(in1 := "SYSTEM_DATA_RETAIN".Detect_Vevtor_1, in2 := 1)
      Contact( "SS Limit 2 Tranfer2" )
      wire#w8
      P_Trig( "Edge_94" )
      S_Coil( "Tranfer_2"."Jog+" )
   END_RUNG
   RUNG wire#w7
      { S7_Templates := "SrcType := Int" } EQ_Contact(in1 := "SYSTEM_DATA_RETAIN".Detect_Vevtor_1, in2 := 2)
      I_Contact( "SS Limit 1 Tranfer2" )
   END_RUNG wire#w8
   RUNG wire#w8
      N_Trig( "Edge_95" )
      R_Coil( "Tranfer_2"."Jog+" )
   END_RUNG
   RUNG wire#w6
      Contact( "Manual_Jog_BW_TF2" )
      wire#w9
      { S7_Templates := "SrcType := Int" } EQ_Contact(in1 := "SYSTEM_DATA_RETAIN".Detect_Vevtor_1, in2 := 1)
      I_Contact( "SS Limit 1 Tranfer2" )
      wire#w10
      P_Trig( "Edge_96" )
      S_Coil( "Tranfer_2"."Jog-" )
   END_RUNG
   RUNG wire#w9
      { S7_Templates := "SrcType := Int" } EQ_Contact(in1 := "SYSTEM_DATA_RETAIN".Detect_Vevtor_1, in2 := 2)
      Contact( "SS Limit 2 Tranfer2" )
   END_RUNG wire#w10
   RUNG wire#w10
      N_Trig( "Edge_97" )
      R_Coil( "Tranfer_2"."Jog-" )
   END_RUNG
   RUNG wire#powerrail
      Contact( "MANUAL_STATE" )
      wire#w11
      Contact( "Manual_Run_FW_TF1" )
      wire#w12
      { S7_Templates := "SrcType := Int" } EQ_Contact(in1 := "SYSTEM_DATA_RETAIN".Detect_Vevtor, in2 := 1)
      Contact( "SS Limit 2 Tranfer1" )
      wire#w13
      P_Trig( "Edge_110" )
      S_Coil( "Tranfer_1".Run_FW )
   END_RUNG
   RUNG wire#w12
      { S7_Templates := "SrcType := Int" } EQ_Contact(in1 := "SYSTEM_DATA_RETAIN".Detect_Vevtor, in2 := 2)
      I_Contact( "SS Limit 1 Tranfer1" )
   END_RUNG wire#w13
   RUNG wire#w13
      N_Trig( "Edge_111" )
      R_Coil( "Tranfer_1".Run_FW )
   END_RUNG
   RUNG wire#w11
      Contact( "Manual_Run_BW_TF1" )
      wire#w14
      { S7_Templates := "SrcType := Int" } EQ_Contact(in1 := "SYSTEM_DATA_RETAIN".Detect_Vevtor, in2 := 1)
      I_Contact( "SS Limit 1 Tranfer1" )
      wire#w15
      P_Trig( "Edge_112" )
      S_Coil( "Tranfer_1".Run_BW )
   END_RUNG
   RUNG wire#w14
      { S7_Templates := "SrcType := Int" } EQ_Contact(in1 := "SYSTEM_DATA_RETAIN".Detect_Vevtor, in2 := 2)
      Contact( "SS Limit 2 Tranfer1" )
   END_RUNG wire#w15
   RUNG wire#w15
      N_Trig( "Edge_113" )
      R_Coil( "Tranfer_1".Run_BW )
   END_RUNG
   RUNG wire#powerrail
      Contact( "MANUAL_STATE" )
      wire#w16
      Contact( "Manual_Run_FW_TF2" )
      wire#w17
      { S7_Templates := "SrcType := Int" } EQ_Contact(in1 := "SYSTEM_DATA_RETAIN".Detect_Vevtor_1, in2 := 1)
      Contact( "SS Limit 2 Tranfer2" )
      wire#w18
      P_Trig( "Edge_126" )
      S_Coil( "Tranfer_2".Run_FW )
   END_RUNG
   RUNG wire#w17
      { S7_Templates := "SrcType := Int" } EQ_Contact(in1 := "SYSTEM_DATA_RETAIN".Detect_Vevtor_1, in2 := 2)
      I_Contact( "SS Limit 1 Tranfer2" )
   END_RUNG wire#w18
   RUNG wire#w18
      N_Trig( "Edge_127" )
      R_Coil( "Tranfer_2".Run_FW )
   END_RUNG
   RUNG wire#w16
      Contact( "Manual_Run_BW_TF2" )
      wire#w19
      { S7_Templates := "SrcType := Int" } EQ_Contact(in1 := "SYSTEM_DATA_RETAIN".Detect_Vevtor_1, in2 := 1)
      I_Contact( "SS Limit 1 Tranfer2" )
      wire#w20
      P_Trig( "Edge_128" )
      S_Coil( "Tranfer_2".Run_BW )
   END_RUNG
   RUNG wire#w19
      { S7_Templates := "SrcType := Int" } EQ_Contact(in1 := "SYSTEM_DATA_RETAIN".Detect_Vevtor_1, in2 := 2)
      Contact( "SS Limit 2 Tranfer2" )
   END_RUNG wire#w20
   RUNG wire#w20
      N_Trig( "Edge_129" )
      R_Coil( "Tranfer_2".Run_BW )
   END_RUNG
   // the same network as SCL:
   #_w1 := "Jog_TF_1_FW" AND NOT "Edge_14";   // rising edge of "Jog_TF_1_FW"
   "Edge_14" := "Jog_TF_1_FW";
   IF #_w1 THEN "Tranfer_1"."Jog+" := TRUE; END_IF;
   #_w2 := NOT "Jog_TF_1_FW" AND "Edge_15";   // falling edge of "Jog_TF_1_FW"
   "Edge_15" := "Jog_TF_1_FW";
   IF #_w2 THEN "Tranfer_1"."Jog+" := FALSE; END_IF;
   #_w3 := "Jog_TF_1_BW" AND NOT "Edge_16";   // rising edge of "Jog_TF_1_BW"
   "Edge_16" := "Jog_TF_1_BW";
   IF #_w3 THEN "Tranfer_1"."Jog-" := TRUE; END_IF;
   #_w4 := NOT "Jog_TF_1_BW" AND "Edge_17";   // falling edge of "Jog_TF_1_BW"
   "Edge_17" := "Jog_TF_1_BW";
   IF #_w4 THEN "Tranfer_1"."Jog-" := FALSE; END_IF;
   #_w5 := "Jog_TF_2_FW" AND NOT "Edge_18";   // rising edge of "Jog_TF_2_FW"
   "Edge_18" := "Jog_TF_2_FW";
   IF #_w5 THEN "Tranfer_2"."Jog+" := TRUE; END_IF;
   #_w6 := NOT "Jog_TF_2_FW" AND "Edge_19";   // falling edge of "Jog_TF_2_FW"
   "Edge_19" := "Jog_TF_2_FW";
   IF #_w6 THEN "Tranfer_2"."Jog+" := FALSE; END_IF;
   #_w7 := "Jog_TF_2_BW" AND NOT "Edge_20";   // rising edge of "Jog_TF_2_BW"
   "Edge_20" := "Jog_TF_2_BW";
   IF #_w7 THEN "Tranfer_2"."Jog-" := TRUE; END_IF;
   #_w8 := NOT "Jog_TF_2_BW" AND "Edge_21";   // falling edge of "Jog_TF_2_BW"
   "Edge_21" := "Jog_TF_2_BW";
   IF #_w8 THEN "Tranfer_2"."Jog-" := FALSE; END_IF;
   #_w9 := "Run_TF_1_FW" AND NOT "Edge_22";   // rising edge of "Run_TF_1_FW"
   "Edge_22" := "Run_TF_1_FW";
   IF #_w9 THEN "Tranfer_1".Run_FW := TRUE; END_IF;
   #_w10 := NOT "Run_TF_1_FW" AND "Edge_23";   // falling edge of "Run_TF_1_FW"
   "Edge_23" := "Run_TF_1_FW";
   IF #_w10 THEN "Tranfer_1".Run_FW := FALSE; END_IF;
   #_w11 := "Run_TF_1_BW" AND NOT "Edge_24";   // rising edge of "Run_TF_1_BW"
   "Edge_24" := "Run_TF_1_BW";
   IF #_w11 THEN "Tranfer_1".Run_BW := TRUE; END_IF;
   #_w12 := NOT "Run_TF_1_BW" AND "Edge_25";   // falling edge of "Run_TF_1_BW"
   "Edge_25" := "Run_TF_1_BW";
   IF #_w12 THEN "Tranfer_1".Run_BW := FALSE; END_IF;
   #_w13 := "Run_TF_2_FW" AND NOT "Edge_26";   // rising edge of "Run_TF_2_FW"
   "Edge_26" := "Run_TF_2_FW";
   IF #_w13 THEN "Tranfer_2".Run_FW := TRUE; END_IF;
   #_w14 := NOT "Run_TF_2_FW" AND "Edge_27";   // falling edge of "Run_TF_2_FW"
   "Edge_27" := "Run_TF_2_FW";
   IF #_w14 THEN "Tranfer_2".Run_FW := FALSE; END_IF;
   #_w15 := "Run_TF_2_BW" AND NOT "Edge_28";   // rising edge of "Run_TF_2_BW"
   "Edge_28" := "Run_TF_2_BW";
   IF #_w15 THEN "Tranfer_2".Run_BW := TRUE; END_IF;
   #_w16 := NOT "Run_TF_2_BW" AND "Edge_29";   // falling edge of "Run_TF_2_BW"
   "Edge_29" := "Run_TF_2_BW";
   IF #_w16 THEN "Tranfer_2".Run_BW := FALSE; END_IF;
   #_w17 := "MANUAL_STATE" AND "Manual_Jog_FW_TF1" AND ((("SYSTEM_DATA_RETAIN".Detect_Vevtor = 1) AND "SS Limit 2 Tranfer1") OR (("SYSTEM_DATA_RETAIN".Detect_Vevtor = 2) AND NOT "SS Limit 1 Tranfer1"));
   #_w18 := #_w17 AND NOT "Edge_90";   // rising edge
   "Edge_90" := #_w17;
   IF #_w18 THEN "Tranfer_1"."Jog+" := TRUE; END_IF;
   #_w19 := NOT #_w17 AND "Edge_91";   // falling edge
   "Edge_91" := #_w17;
   IF #_w19 THEN "Tranfer_1"."Jog+" := FALSE; END_IF;
   #_w20 := "MANUAL_STATE" AND "Manual_Jog_BW_TF1" AND ((("SYSTEM_DATA_RETAIN".Detect_Vevtor = 1) AND NOT "SS Limit 1 Tranfer1") OR (("SYSTEM_DATA_RETAIN".Detect_Vevtor = 2) AND "SS Limit 2 Tranfer1"));
   #_w21 := #_w20 AND NOT "Edge_92";   // rising edge
   "Edge_92" := #_w20;
   IF #_w21 THEN "Tranfer_1"."Jog-" := TRUE; END_IF;
   #_w22 := NOT #_w20 AND "Edge_93";   // falling edge
   "Edge_93" := #_w20;
   IF #_w22 THEN "Tranfer_1"."Jog-" := FALSE; END_IF;
   #_w23 := "MANUAL_STATE" AND "Manual_Jog_FW_TF2" AND ((("SYSTEM_DATA_RETAIN".Detect_Vevtor_1 = 1) AND "SS Limit 2 Tranfer2") OR (("SYSTEM_DATA_RETAIN".Detect_Vevtor_1 = 2) AND NOT "SS Limit 1 Tranfer2"));
   #_w24 := #_w23 AND NOT "Edge_94";   // rising edge
   "Edge_94" := #_w23;
   IF #_w24 THEN "Tranfer_2"."Jog+" := TRUE; END_IF;
   #_w25 := NOT #_w23 AND "Edge_95";   // falling edge
   "Edge_95" := #_w23;
   IF #_w25 THEN "Tranfer_2"."Jog+" := FALSE; END_IF;
   #_w26 := "MANUAL_STATE" AND "Manual_Jog_BW_TF2" AND ((("SYSTEM_DATA_RETAIN".Detect_Vevtor_1 = 1) AND NOT "SS Limit 1 Tranfer2") OR (("SYSTEM_DATA_RETAIN".Detect_Vevtor_1 = 2) AND "SS Limit 2 Tranfer2"));
   #_w27 := #_w26 AND NOT "Edge_96";   // rising edge
   "Edge_96" := #_w26;
   IF #_w27 THEN "Tranfer_2"."Jog-" := TRUE; END_IF;
   #_w28 := NOT #_w26 AND "Edge_97";   // falling edge
   "Edge_97" := #_w26;
   IF #_w28 THEN "Tranfer_2"."Jog-" := FALSE; END_IF;
   #_w29 := "MANUAL_STATE" AND "Manual_Run_FW_TF1" AND ((("SYSTEM_DATA_RETAIN".Detect_Vevtor = 1) AND "SS Limit 2 Tranfer1") OR (("SYSTEM_DATA_RETAIN".Detect_Vevtor = 2) AND NOT "SS Limit 1 Tranfer1"));
   #_w30 := #_w29 AND NOT "Edge_110";   // rising edge
   "Edge_110" := #_w29;
   IF #_w30 THEN "Tranfer_1".Run_FW := TRUE; END_IF;
   #_w31 := NOT #_w29 AND "Edge_111";   // falling edge
   "Edge_111" := #_w29;
   IF #_w31 THEN "Tranfer_1".Run_FW := FALSE; END_IF;
   #_w32 := "MANUAL_STATE" AND "Manual_Run_BW_TF1" AND ((("SYSTEM_DATA_RETAIN".Detect_Vevtor = 1) AND NOT "SS Limit 1 Tranfer1") OR (("SYSTEM_DATA_RETAIN".Detect_Vevtor = 2) AND "SS Limit 2 Tranfer1"));
   #_w33 := #_w32 AND NOT "Edge_112";   // rising edge
   "Edge_112" := #_w32;
   IF #_w33 THEN "Tranfer_1".Run_BW := TRUE; END_IF;
   #_w34 := NOT #_w32 AND "Edge_113";   // falling edge
   "Edge_113" := #_w32;
   IF #_w34 THEN "Tranfer_1".Run_BW := FALSE; END_IF;
   #_w35 := "MANUAL_STATE" AND "Manual_Run_FW_TF2" AND ((("SYSTEM_DATA_RETAIN".Detect_Vevtor_1 = 1) AND "SS Limit 2 Tranfer2") OR (("SYSTEM_DATA_RETAIN".Detect_Vevtor_1 = 2) AND NOT "SS Limit 1 Tranfer2"));
   #_w36 := #_w35 AND NOT "Edge_126";   // rising edge
   "Edge_126" := #_w35;
   IF #_w36 THEN "Tranfer_2".Run_FW := TRUE; END_IF;
   #_w37 := NOT #_w35 AND "Edge_127";   // falling edge
   "Edge_127" := #_w35;
   IF #_w37 THEN "Tranfer_2".Run_FW := FALSE; END_IF;
   #_w38 := "MANUAL_STATE" AND "Manual_Run_BW_TF2" AND ((("SYSTEM_DATA_RETAIN".Detect_Vevtor_1 = 1) AND NOT "SS Limit 1 Tranfer2") OR (("SYSTEM_DATA_RETAIN".Detect_Vevtor_1 = 2) AND "SS Limit 2 Tranfer2"));
   #_w39 := #_w38 AND NOT "Edge_128";   // rising edge
   "Edge_128" := #_w38;
   IF #_w39 THEN "Tranfer_2".Run_BW := TRUE; END_IF;
   #_w40 := NOT #_w38 AND "Edge_129";   // falling edge
   "Edge_129" := #_w38;
   IF #_w40 THEN "Tranfer_2".Run_BW := FALSE; END_IF;
END_REGION

REGION Network 19: Setting Config Tranfer
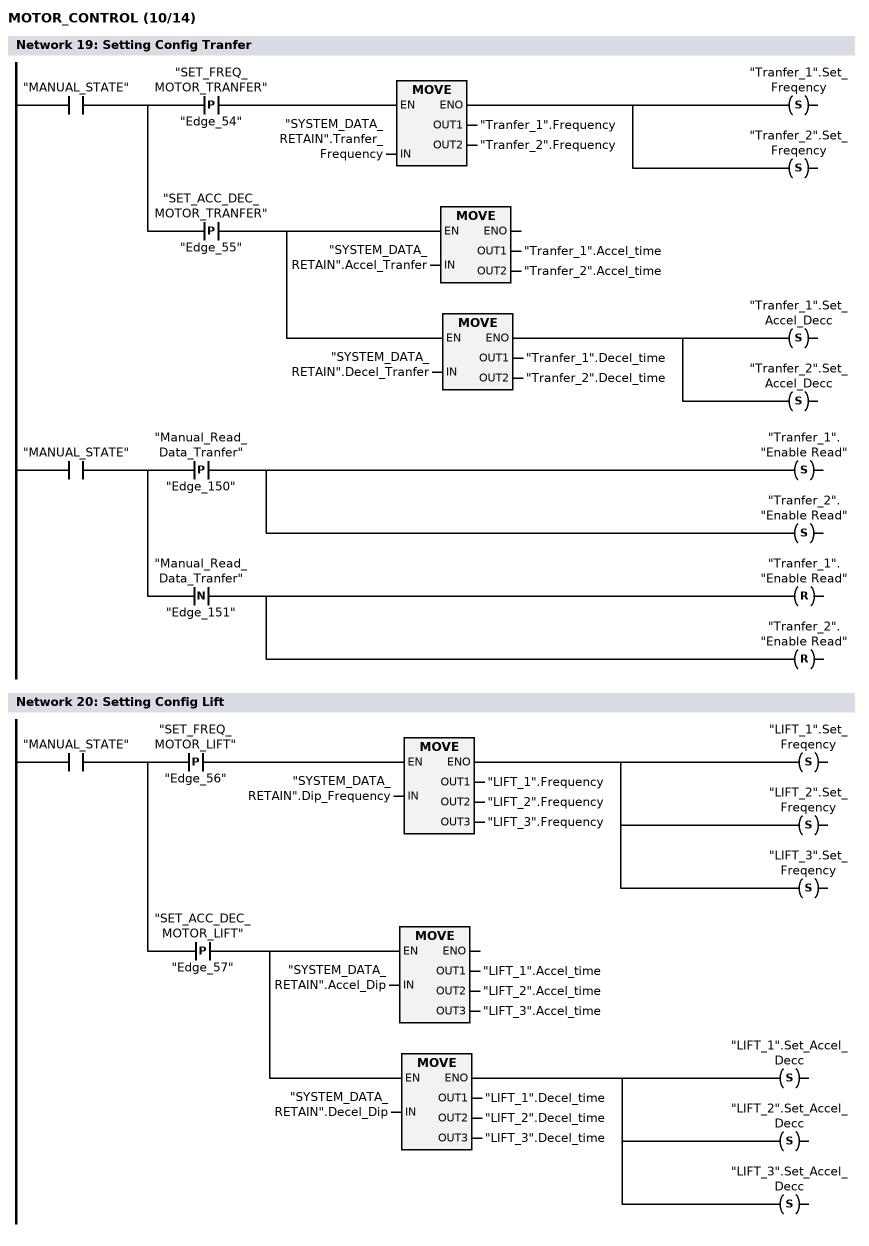
   RUNG wire#powerrail
      Contact( "MANUAL_STATE" )
      wire#w1
      P_Contact(operand := "SET_FREQ_MOTOR_TRANFER", bit := "Edge_54")
      { S7_GenerateENO := "TRUE" } Move(in := "SYSTEM_DATA_RETAIN".Tranfer_Frequency, out1 => "Tranfer_1".Frequency, out2 => "Tranfer_2".Frequency)
      wire#w2
      S_Coil( "Tranfer_1".Set_Freqency )
   END_RUNG
   RUNG wire#w2
      S_Coil( "Tranfer_2".Set_Freqency )
   END_RUNG
   RUNG wire#w1
      P_Contact(operand := "SET_ACC_DEC_MOTOR_TRANFER", bit := "Edge_55")
      wire#w3
      { S7_GenerateENO := "TRUE" } Move(in := "SYSTEM_DATA_RETAIN".Accel_Tranfer, out1 => "Tranfer_1".Accel_time, out2 => "Tranfer_2".Accel_time)
   END_RUNG
   RUNG wire#w3
      { S7_GenerateENO := "TRUE" } Move(in := "SYSTEM_DATA_RETAIN".Decel_Tranfer, out1 => "Tranfer_1".Decel_time, out2 => "Tranfer_2".Decel_time)
      wire#w4
      S_Coil( "Tranfer_1".Set_Accel_Decc )
   END_RUNG
   RUNG wire#w4
      S_Coil( "Tranfer_2".Set_Accel_Decc )
   END_RUNG
   RUNG wire#powerrail
      Contact( "MANUAL_STATE" )
      wire#w5
      P_Contact(operand := "Manual_Read_Data_Tranfer", bit := "Edge_150")
      wire#w6
      S_Coil( "Tranfer_1"."Enable Read" )
   END_RUNG
   RUNG wire#w6
      S_Coil( "Tranfer_2"."Enable Read" )
   END_RUNG
   RUNG wire#w5
      N_Contact(operand := "Manual_Read_Data_Tranfer", bit := "Edge_151")
      wire#w7
      R_Coil( "Tranfer_1"."Enable Read" )
   END_RUNG
   RUNG wire#w7
      R_Coil( "Tranfer_2"."Enable Read" )
   END_RUNG
   // the same network as SCL:
   // ENO of a box is taken as its EN; it also drops when the box reports an error
   #_w1 := "MANUAL_STATE" AND "SET_FREQ_MOTOR_TRANFER" AND NOT "Edge_54";   // rising edge of "SET_FREQ_MOTOR_TRANFER"
   "Edge_54" := "SET_FREQ_MOTOR_TRANFER";
   IF #_w1 THEN
       "Tranfer_1".Frequency := "SYSTEM_DATA_RETAIN".Tranfer_Frequency;
       "Tranfer_2".Frequency := "SYSTEM_DATA_RETAIN".Tranfer_Frequency;
       "Tranfer_1".Set_Freqency := TRUE;
       "Tranfer_2".Set_Freqency := TRUE;
   END_IF;
   #_w2 := "MANUAL_STATE" AND "SET_ACC_DEC_MOTOR_TRANFER" AND NOT "Edge_55";   // rising edge of "SET_ACC_DEC_MOTOR_TRANFER"
   "Edge_55" := "SET_ACC_DEC_MOTOR_TRANFER";
   IF #_w2 THEN
       "Tranfer_1".Accel_time := "SYSTEM_DATA_RETAIN".Accel_Tranfer;
       "Tranfer_2".Accel_time := "SYSTEM_DATA_RETAIN".Accel_Tranfer;
       "Tranfer_1".Decel_time := "SYSTEM_DATA_RETAIN".Decel_Tranfer;
       "Tranfer_2".Decel_time := "SYSTEM_DATA_RETAIN".Decel_Tranfer;
       "Tranfer_1".Set_Accel_Decc := TRUE;
       "Tranfer_2".Set_Accel_Decc := TRUE;
   END_IF;
   #_w3 := "MANUAL_STATE" AND "Manual_Read_Data_Tranfer" AND NOT "Edge_150";   // rising edge of "Manual_Read_Data_Tranfer"
   "Edge_150" := "Manual_Read_Data_Tranfer";
   IF #_w3 THEN
       "Tranfer_1"."Enable Read" := TRUE;
       "Tranfer_2"."Enable Read" := TRUE;
   END_IF;
   #_w4 := "MANUAL_STATE" AND NOT "Manual_Read_Data_Tranfer" AND "Edge_151";   // falling edge of "Manual_Read_Data_Tranfer"
   "Edge_151" := "Manual_Read_Data_Tranfer";
   IF #_w4 THEN
       "Tranfer_1"."Enable Read" := FALSE;
       "Tranfer_2"."Enable Read" := FALSE;
   END_IF;
END_REGION

REGION Network 20: Setting Config Lift
   RUNG wire#powerrail
      Contact( "MANUAL_STATE" )
      wire#w1
      P_Contact(operand := "SET_FREQ_MOTOR_LIFT", bit := "Edge_56")
      { S7_GenerateENO := "TRUE" } Move(in := "SYSTEM_DATA_RETAIN".Dip_Frequency, out1 => "LIFT_1".Frequency, out2 => "LIFT_2".Frequency, out3 => "LIFT_3".Frequency)
      wire#w2
      S_Coil( "LIFT_1".Set_Freqency )
   END_RUNG
   RUNG wire#w2
      S_Coil( "LIFT_2".Set_Freqency )
   END_RUNG
   RUNG wire#w2
      S_Coil( "LIFT_3".Set_Freqency )
   END_RUNG
   RUNG wire#w1
      P_Contact(operand := "SET_ACC_DEC_MOTOR_LIFT", bit := "Edge_57")
      wire#w3
      { S7_GenerateENO := "TRUE" } Move(in := "SYSTEM_DATA_RETAIN".Accel_Dip, out1 => "LIFT_1".Accel_time, out2 => "LIFT_2".Accel_time, out3 => "LIFT_3".Accel_time)
   END_RUNG
   RUNG wire#w3
      { S7_GenerateENO := "TRUE" } Move(in := "SYSTEM_DATA_RETAIN".Decel_Dip, out1 => "LIFT_1".Decel_time, out2 => "LIFT_2".Decel_time, out3 => "LIFT_3".Decel_time)
      wire#w4
      S_Coil( "LIFT_1".Set_Accel_Decc )
   END_RUNG
   RUNG wire#w4
      S_Coil( "LIFT_2".Set_Accel_Decc )
   END_RUNG
   RUNG wire#w4
      S_Coil( "LIFT_3".Set_Accel_Decc )
   END_RUNG
   // the same network as SCL:
   // ENO of a box is taken as its EN; it also drops when the box reports an error
   #_w1 := "MANUAL_STATE" AND "SET_FREQ_MOTOR_LIFT" AND NOT "Edge_56";   // rising edge of "SET_FREQ_MOTOR_LIFT"
   "Edge_56" := "SET_FREQ_MOTOR_LIFT";
   IF #_w1 THEN
       "LIFT_1".Frequency := "SYSTEM_DATA_RETAIN".Dip_Frequency;
       "LIFT_2".Frequency := "SYSTEM_DATA_RETAIN".Dip_Frequency;
       "LIFT_3".Frequency := "SYSTEM_DATA_RETAIN".Dip_Frequency;
       "LIFT_1".Set_Freqency := TRUE;
       "LIFT_2".Set_Freqency := TRUE;
       "LIFT_3".Set_Freqency := TRUE;
   END_IF;
   #_w2 := "MANUAL_STATE" AND "SET_ACC_DEC_MOTOR_LIFT" AND NOT "Edge_57";   // rising edge of "SET_ACC_DEC_MOTOR_LIFT"
   "Edge_57" := "SET_ACC_DEC_MOTOR_LIFT";
   IF #_w2 THEN
       "LIFT_1".Accel_time := "SYSTEM_DATA_RETAIN".Accel_Dip;
       "LIFT_2".Accel_time := "SYSTEM_DATA_RETAIN".Accel_Dip;
       "LIFT_3".Accel_time := "SYSTEM_DATA_RETAIN".Accel_Dip;
       "LIFT_1".Decel_time := "SYSTEM_DATA_RETAIN".Decel_Dip;
       "LIFT_2".Decel_time := "SYSTEM_DATA_RETAIN".Decel_Dip;
       "LIFT_3".Decel_time := "SYSTEM_DATA_RETAIN".Decel_Dip;
       "LIFT_1".Set_Accel_Decc := TRUE;
       "LIFT_2".Set_Accel_Decc := TRUE;
       "LIFT_3".Set_Accel_Decc := TRUE;
   END_IF;
END_REGION

REGION Network 21: JOG / RUN LIFT 1
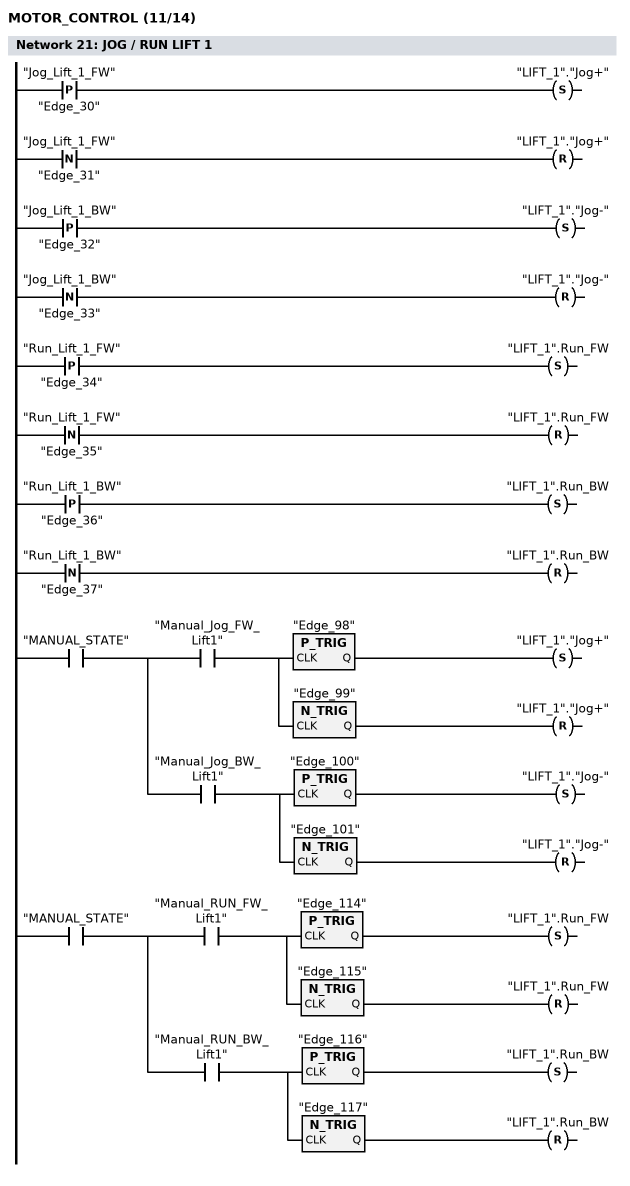
   RUNG wire#powerrail
      P_Contact(operand := "Jog_Lift_1_FW", bit := "Edge_30")
      S_Coil( "LIFT_1"."Jog+" )
   END_RUNG
   RUNG wire#powerrail
      N_Contact(operand := "Jog_Lift_1_FW", bit := "Edge_31")
      R_Coil( "LIFT_1"."Jog+" )
   END_RUNG
   RUNG wire#powerrail
      P_Contact(operand := "Jog_Lift_1_BW", bit := "Edge_32")
      S_Coil( "LIFT_1"."Jog-" )
   END_RUNG
   RUNG wire#powerrail
      N_Contact(operand := "Jog_Lift_1_BW", bit := "Edge_33")
      R_Coil( "LIFT_1"."Jog-" )
   END_RUNG
   RUNG wire#powerrail
      P_Contact(operand := "Run_Lift_1_FW", bit := "Edge_34")
      S_Coil( "LIFT_1".Run_FW )
   END_RUNG
   RUNG wire#powerrail
      N_Contact(operand := "Run_Lift_1_FW", bit := "Edge_35")
      R_Coil( "LIFT_1".Run_FW )
   END_RUNG
   RUNG wire#powerrail
      P_Contact(operand := "Run_Lift_1_BW", bit := "Edge_36")
      S_Coil( "LIFT_1".Run_BW )
   END_RUNG
   RUNG wire#powerrail
      N_Contact(operand := "Run_Lift_1_BW", bit := "Edge_37")
      R_Coil( "LIFT_1".Run_BW )
   END_RUNG
   RUNG wire#powerrail
      Contact( "MANUAL_STATE" )
      wire#w1
      Contact( "Manual_Jog_FW_Lift1" )
      wire#w2
      P_Trig( "Edge_98" )
      S_Coil( "LIFT_1"."Jog+" )
   END_RUNG
   RUNG wire#w2
      N_Trig( "Edge_99" )
      R_Coil( "LIFT_1"."Jog+" )
   END_RUNG
   RUNG wire#w1
      Contact( "Manual_Jog_BW_Lift1" )
      wire#w3
      P_Trig( "Edge_100" )
      S_Coil( "LIFT_1"."Jog-" )
   END_RUNG
   RUNG wire#w3
      N_Trig( "Edge_101" )
      R_Coil( "LIFT_1"."Jog-" )
   END_RUNG
   RUNG wire#powerrail
      Contact( "MANUAL_STATE" )
      wire#w4
      Contact( "Manual_RUN_FW_Lift1" )
      wire#w5
      P_Trig( "Edge_114" )
      S_Coil( "LIFT_1".Run_FW )
   END_RUNG
   RUNG wire#w5
      N_Trig( "Edge_115" )
      R_Coil( "LIFT_1".Run_FW )
   END_RUNG
   RUNG wire#w4
      Contact( "Manual_RUN_BW_Lift1" )
      wire#w6
      P_Trig( "Edge_116" )
      S_Coil( "LIFT_1".Run_BW )
   END_RUNG
   RUNG wire#w6
      N_Trig( "Edge_117" )
      R_Coil( "LIFT_1".Run_BW )
   END_RUNG
   // the same network as SCL:
   #_w1 := "Jog_Lift_1_FW" AND NOT "Edge_30";   // rising edge of "Jog_Lift_1_FW"
   "Edge_30" := "Jog_Lift_1_FW";
   IF #_w1 THEN "LIFT_1"."Jog+" := TRUE; END_IF;
   #_w2 := NOT "Jog_Lift_1_FW" AND "Edge_31";   // falling edge of "Jog_Lift_1_FW"
   "Edge_31" := "Jog_Lift_1_FW";
   IF #_w2 THEN "LIFT_1"."Jog+" := FALSE; END_IF;
   #_w3 := "Jog_Lift_1_BW" AND NOT "Edge_32";   // rising edge of "Jog_Lift_1_BW"
   "Edge_32" := "Jog_Lift_1_BW";
   IF #_w3 THEN "LIFT_1"."Jog-" := TRUE; END_IF;
   #_w4 := NOT "Jog_Lift_1_BW" AND "Edge_33";   // falling edge of "Jog_Lift_1_BW"
   "Edge_33" := "Jog_Lift_1_BW";
   IF #_w4 THEN "LIFT_1"."Jog-" := FALSE; END_IF;
   #_w5 := "Run_Lift_1_FW" AND NOT "Edge_34";   // rising edge of "Run_Lift_1_FW"
   "Edge_34" := "Run_Lift_1_FW";
   IF #_w5 THEN "LIFT_1".Run_FW := TRUE; END_IF;
   #_w6 := NOT "Run_Lift_1_FW" AND "Edge_35";   // falling edge of "Run_Lift_1_FW"
   "Edge_35" := "Run_Lift_1_FW";
   IF #_w6 THEN "LIFT_1".Run_FW := FALSE; END_IF;
   #_w7 := "Run_Lift_1_BW" AND NOT "Edge_36";   // rising edge of "Run_Lift_1_BW"
   "Edge_36" := "Run_Lift_1_BW";
   IF #_w7 THEN "LIFT_1".Run_BW := TRUE; END_IF;
   #_w8 := NOT "Run_Lift_1_BW" AND "Edge_37";   // falling edge of "Run_Lift_1_BW"
   "Edge_37" := "Run_Lift_1_BW";
   IF #_w8 THEN "LIFT_1".Run_BW := FALSE; END_IF;
   #_w9 := "MANUAL_STATE" AND "Manual_Jog_FW_Lift1";
   #_w10 := #_w9 AND NOT "Edge_98";   // rising edge
   "Edge_98" := #_w9;
   IF #_w10 THEN "LIFT_1"."Jog+" := TRUE; END_IF;
   #_w11 := NOT #_w9 AND "Edge_99";   // falling edge
   "Edge_99" := #_w9;
   IF #_w11 THEN "LIFT_1"."Jog+" := FALSE; END_IF;
   #_w12 := "MANUAL_STATE" AND "Manual_Jog_BW_Lift1";
   #_w13 := #_w12 AND NOT "Edge_100";   // rising edge
   "Edge_100" := #_w12;
   IF #_w13 THEN "LIFT_1"."Jog-" := TRUE; END_IF;
   #_w14 := NOT #_w12 AND "Edge_101";   // falling edge
   "Edge_101" := #_w12;
   IF #_w14 THEN "LIFT_1"."Jog-" := FALSE; END_IF;
   #_w15 := "MANUAL_STATE" AND "Manual_RUN_FW_Lift1";
   #_w16 := #_w15 AND NOT "Edge_114";   // rising edge
   "Edge_114" := #_w15;
   IF #_w16 THEN "LIFT_1".Run_FW := TRUE; END_IF;
   #_w17 := NOT #_w15 AND "Edge_115";   // falling edge
   "Edge_115" := #_w15;
   IF #_w17 THEN "LIFT_1".Run_FW := FALSE; END_IF;
   #_w18 := "MANUAL_STATE" AND "Manual_RUN_BW_Lift1";
   #_w19 := #_w18 AND NOT "Edge_116";   // rising edge
   "Edge_116" := #_w18;
   IF #_w19 THEN "LIFT_1".Run_BW := TRUE; END_IF;
   #_w20 := NOT #_w18 AND "Edge_117";   // falling edge
   "Edge_117" := #_w18;
   IF #_w20 THEN "LIFT_1".Run_BW := FALSE; END_IF;
END_REGION

REGION Network 22: JOG / RUN LIFt 2
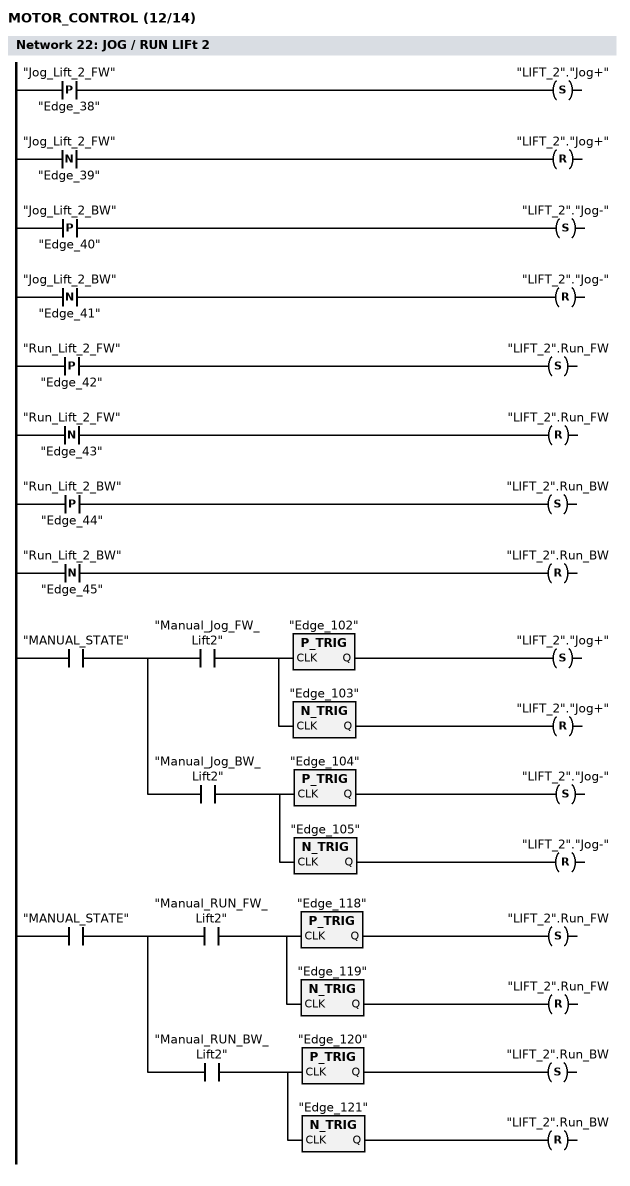
   RUNG wire#powerrail
      P_Contact(operand := "Jog_Lift_2_FW", bit := "Edge_38")
      S_Coil( "LIFT_2"."Jog+" )
   END_RUNG
   RUNG wire#powerrail
      N_Contact(operand := "Jog_Lift_2_FW", bit := "Edge_39")
      R_Coil( "LIFT_2"."Jog+" )
   END_RUNG
   RUNG wire#powerrail
      P_Contact(operand := "Jog_Lift_2_BW", bit := "Edge_40")
      S_Coil( "LIFT_2"."Jog-" )
   END_RUNG
   RUNG wire#powerrail
      N_Contact(operand := "Jog_Lift_2_BW", bit := "Edge_41")
      R_Coil( "LIFT_2"."Jog-" )
   END_RUNG
   RUNG wire#powerrail
      P_Contact(operand := "Run_Lift_2_FW", bit := "Edge_42")
      S_Coil( "LIFT_2".Run_FW )
   END_RUNG
   RUNG wire#powerrail
      N_Contact(operand := "Run_Lift_2_FW", bit := "Edge_43")
      R_Coil( "LIFT_2".Run_FW )
   END_RUNG
   RUNG wire#powerrail
      P_Contact(operand := "Run_Lift_2_BW", bit := "Edge_44")
      S_Coil( "LIFT_2".Run_BW )
   END_RUNG
   RUNG wire#powerrail
      N_Contact(operand := "Run_Lift_2_BW", bit := "Edge_45")
      R_Coil( "LIFT_2".Run_BW )
   END_RUNG
   RUNG wire#powerrail
      Contact( "MANUAL_STATE" )
      wire#w1
      Contact( "Manual_Jog_FW_Lift2" )
      wire#w2
      P_Trig( "Edge_102" )
      S_Coil( "LIFT_2"."Jog+" )
   END_RUNG
   RUNG wire#w2
      N_Trig( "Edge_103" )
      R_Coil( "LIFT_2"."Jog+" )
   END_RUNG
   RUNG wire#w1
      Contact( "Manual_Jog_BW_Lift2" )
      wire#w3
      P_Trig( "Edge_104" )
      S_Coil( "LIFT_2"."Jog-" )
   END_RUNG
   RUNG wire#w3
      N_Trig( "Edge_105" )
      R_Coil( "LIFT_2"."Jog-" )
   END_RUNG
   RUNG wire#powerrail
      Contact( "MANUAL_STATE" )
      wire#w4
      Contact( "Manual_RUN_FW_Lift2" )
      wire#w5
      P_Trig( "Edge_118" )
      S_Coil( "LIFT_2".Run_FW )
   END_RUNG
   RUNG wire#w5
      N_Trig( "Edge_119" )
      R_Coil( "LIFT_2".Run_FW )
   END_RUNG
   RUNG wire#w4
      Contact( "Manual_RUN_BW_Lift2" )
      wire#w6
      P_Trig( "Edge_120" )
      S_Coil( "LIFT_2".Run_BW )
   END_RUNG
   RUNG wire#w6
      N_Trig( "Edge_121" )
      R_Coil( "LIFT_2".Run_BW )
   END_RUNG
   // the same network as SCL:
   #_w1 := "Jog_Lift_2_FW" AND NOT "Edge_38";   // rising edge of "Jog_Lift_2_FW"
   "Edge_38" := "Jog_Lift_2_FW";
   IF #_w1 THEN "LIFT_2"."Jog+" := TRUE; END_IF;
   #_w2 := NOT "Jog_Lift_2_FW" AND "Edge_39";   // falling edge of "Jog_Lift_2_FW"
   "Edge_39" := "Jog_Lift_2_FW";
   IF #_w2 THEN "LIFT_2"."Jog+" := FALSE; END_IF;
   #_w3 := "Jog_Lift_2_BW" AND NOT "Edge_40";   // rising edge of "Jog_Lift_2_BW"
   "Edge_40" := "Jog_Lift_2_BW";
   IF #_w3 THEN "LIFT_2"."Jog-" := TRUE; END_IF;
   #_w4 := NOT "Jog_Lift_2_BW" AND "Edge_41";   // falling edge of "Jog_Lift_2_BW"
   "Edge_41" := "Jog_Lift_2_BW";
   IF #_w4 THEN "LIFT_2"."Jog-" := FALSE; END_IF;
   #_w5 := "Run_Lift_2_FW" AND NOT "Edge_42";   // rising edge of "Run_Lift_2_FW"
   "Edge_42" := "Run_Lift_2_FW";
   IF #_w5 THEN "LIFT_2".Run_FW := TRUE; END_IF;
   #_w6 := NOT "Run_Lift_2_FW" AND "Edge_43";   // falling edge of "Run_Lift_2_FW"
   "Edge_43" := "Run_Lift_2_FW";
   IF #_w6 THEN "LIFT_2".Run_FW := FALSE; END_IF;
   #_w7 := "Run_Lift_2_BW" AND NOT "Edge_44";   // rising edge of "Run_Lift_2_BW"
   "Edge_44" := "Run_Lift_2_BW";
   IF #_w7 THEN "LIFT_2".Run_BW := TRUE; END_IF;
   #_w8 := NOT "Run_Lift_2_BW" AND "Edge_45";   // falling edge of "Run_Lift_2_BW"
   "Edge_45" := "Run_Lift_2_BW";
   IF #_w8 THEN "LIFT_2".Run_BW := FALSE; END_IF;
   #_w9 := "MANUAL_STATE" AND "Manual_Jog_FW_Lift2";
   #_w10 := #_w9 AND NOT "Edge_102";   // rising edge
   "Edge_102" := #_w9;
   IF #_w10 THEN "LIFT_2"."Jog+" := TRUE; END_IF;
   #_w11 := NOT #_w9 AND "Edge_103";   // falling edge
   "Edge_103" := #_w9;
   IF #_w11 THEN "LIFT_2"."Jog+" := FALSE; END_IF;
   #_w12 := "MANUAL_STATE" AND "Manual_Jog_BW_Lift2";
   #_w13 := #_w12 AND NOT "Edge_104";   // rising edge
   "Edge_104" := #_w12;
   IF #_w13 THEN "LIFT_2"."Jog-" := TRUE; END_IF;
   #_w14 := NOT #_w12 AND "Edge_105";   // falling edge
   "Edge_105" := #_w12;
   IF #_w14 THEN "LIFT_2"."Jog-" := FALSE; END_IF;
   #_w15 := "MANUAL_STATE" AND "Manual_RUN_FW_Lift2";
   #_w16 := #_w15 AND NOT "Edge_118";   // rising edge
   "Edge_118" := #_w15;
   IF #_w16 THEN "LIFT_2".Run_FW := TRUE; END_IF;
   #_w17 := NOT #_w15 AND "Edge_119";   // falling edge
   "Edge_119" := #_w15;
   IF #_w17 THEN "LIFT_2".Run_FW := FALSE; END_IF;
   #_w18 := "MANUAL_STATE" AND "Manual_RUN_BW_Lift2";
   #_w19 := #_w18 AND NOT "Edge_120";   // rising edge
   "Edge_120" := #_w18;
   IF #_w19 THEN "LIFT_2".Run_BW := TRUE; END_IF;
   #_w20 := NOT #_w18 AND "Edge_121";   // falling edge
   "Edge_121" := #_w18;
   IF #_w20 THEN "LIFT_2".Run_BW := FALSE; END_IF;
END_REGION

REGION Network 23: JOG / RUN LIFt 3
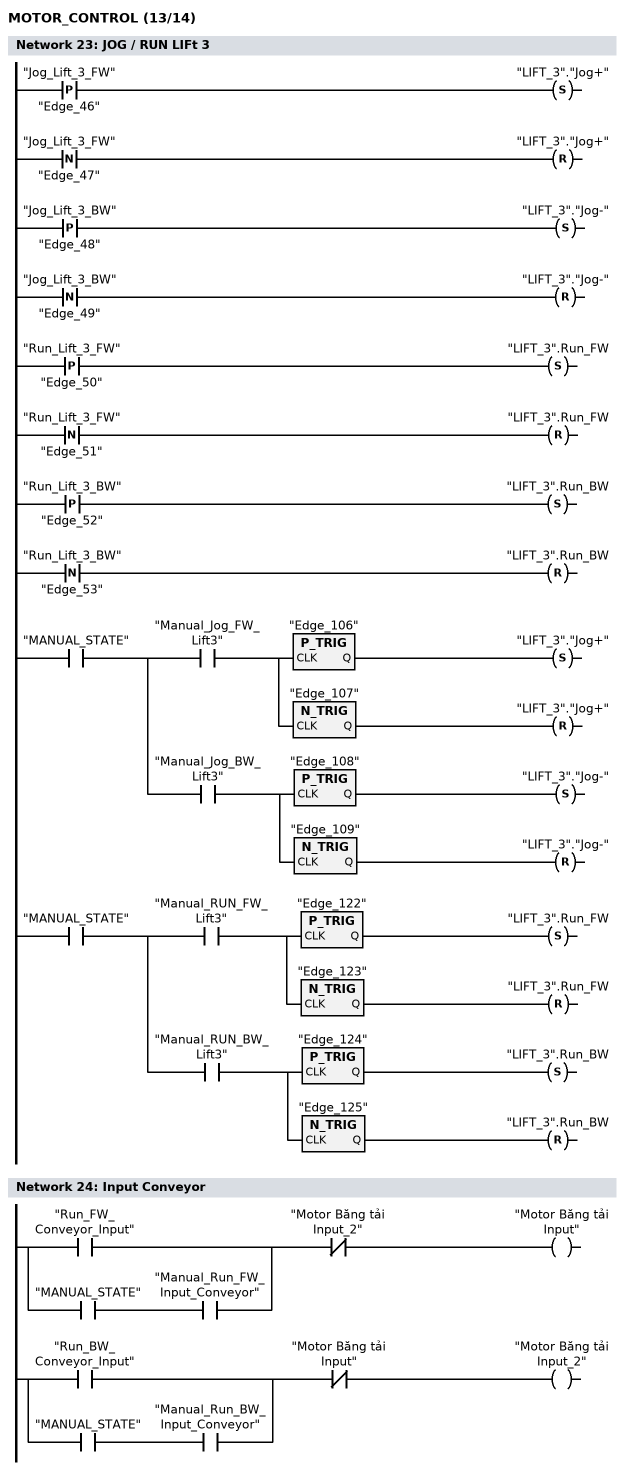
   RUNG wire#powerrail
      P_Contact(operand := "Jog_Lift_3_FW", bit := "Edge_46")
      S_Coil( "LIFT_3"."Jog+" )
   END_RUNG
   RUNG wire#powerrail
      N_Contact(operand := "Jog_Lift_3_FW", bit := "Edge_47")
      R_Coil( "LIFT_3"."Jog+" )
   END_RUNG
   RUNG wire#powerrail
      P_Contact(operand := "Jog_Lift_3_BW", bit := "Edge_48")
      S_Coil( "LIFT_3"."Jog-" )
   END_RUNG
   RUNG wire#powerrail
      N_Contact(operand := "Jog_Lift_3_BW", bit := "Edge_49")
      R_Coil( "LIFT_3"."Jog-" )
   END_RUNG
   RUNG wire#powerrail
      P_Contact(operand := "Run_Lift_3_FW", bit := "Edge_50")
      S_Coil( "LIFT_3".Run_FW )
   END_RUNG
   RUNG wire#powerrail
      N_Contact(operand := "Run_Lift_3_FW", bit := "Edge_51")
      R_Coil( "LIFT_3".Run_FW )
   END_RUNG
   RUNG wire#powerrail
      P_Contact(operand := "Run_Lift_3_BW", bit := "Edge_52")
      S_Coil( "LIFT_3".Run_BW )
   END_RUNG
   RUNG wire#powerrail
      N_Contact(operand := "Run_Lift_3_BW", bit := "Edge_53")
      R_Coil( "LIFT_3".Run_BW )
   END_RUNG
   RUNG wire#powerrail
      Contact( "MANUAL_STATE" )
      wire#w1
      Contact( "Manual_Jog_FW_Lift3" )
      wire#w2
      P_Trig( "Edge_106" )
      S_Coil( "LIFT_3"."Jog+" )
   END_RUNG
   RUNG wire#w2
      N_Trig( "Edge_107" )
      R_Coil( "LIFT_3"."Jog+" )
   END_RUNG
   RUNG wire#w1
      Contact( "Manual_Jog_BW_Lift3" )
      wire#w3
      P_Trig( "Edge_108" )
      S_Coil( "LIFT_3"."Jog-" )
   END_RUNG
   RUNG wire#w3
      N_Trig( "Edge_109" )
      R_Coil( "LIFT_3"."Jog-" )
   END_RUNG
   RUNG wire#powerrail
      Contact( "MANUAL_STATE" )
      wire#w4
      Contact( "Manual_RUN_FW_Lift3" )
      wire#w5
      P_Trig( "Edge_122" )
      S_Coil( "LIFT_3".Run_FW )
   END_RUNG
   RUNG wire#w5
      N_Trig( "Edge_123" )
      R_Coil( "LIFT_3".Run_FW )
   END_RUNG
   RUNG wire#w4
      Contact( "Manual_RUN_BW_Lift3" )
      wire#w6
      P_Trig( "Edge_124" )
      S_Coil( "LIFT_3".Run_BW )
   END_RUNG
   RUNG wire#w6
      N_Trig( "Edge_125" )
      R_Coil( "LIFT_3".Run_BW )
   END_RUNG
   // the same network as SCL:
   #_w1 := "Jog_Lift_3_FW" AND NOT "Edge_46";   // rising edge of "Jog_Lift_3_FW"
   "Edge_46" := "Jog_Lift_3_FW";
   IF #_w1 THEN "LIFT_3"."Jog+" := TRUE; END_IF;
   #_w2 := NOT "Jog_Lift_3_FW" AND "Edge_47";   // falling edge of "Jog_Lift_3_FW"
   "Edge_47" := "Jog_Lift_3_FW";
   IF #_w2 THEN "LIFT_3"."Jog+" := FALSE; END_IF;
   #_w3 := "Jog_Lift_3_BW" AND NOT "Edge_48";   // rising edge of "Jog_Lift_3_BW"
   "Edge_48" := "Jog_Lift_3_BW";
   IF #_w3 THEN "LIFT_3"."Jog-" := TRUE; END_IF;
   #_w4 := NOT "Jog_Lift_3_BW" AND "Edge_49";   // falling edge of "Jog_Lift_3_BW"
   "Edge_49" := "Jog_Lift_3_BW";
   IF #_w4 THEN "LIFT_3"."Jog-" := FALSE; END_IF;
   #_w5 := "Run_Lift_3_FW" AND NOT "Edge_50";   // rising edge of "Run_Lift_3_FW"
   "Edge_50" := "Run_Lift_3_FW";
   IF #_w5 THEN "LIFT_3".Run_FW := TRUE; END_IF;
   #_w6 := NOT "Run_Lift_3_FW" AND "Edge_51";   // falling edge of "Run_Lift_3_FW"
   "Edge_51" := "Run_Lift_3_FW";
   IF #_w6 THEN "LIFT_3".Run_FW := FALSE; END_IF;
   #_w7 := "Run_Lift_3_BW" AND NOT "Edge_52";   // rising edge of "Run_Lift_3_BW"
   "Edge_52" := "Run_Lift_3_BW";
   IF #_w7 THEN "LIFT_3".Run_BW := TRUE; END_IF;
   #_w8 := NOT "Run_Lift_3_BW" AND "Edge_53";   // falling edge of "Run_Lift_3_BW"
   "Edge_53" := "Run_Lift_3_BW";
   IF #_w8 THEN "LIFT_3".Run_BW := FALSE; END_IF;
   #_w9 := "MANUAL_STATE" AND "Manual_Jog_FW_Lift3";
   #_w10 := #_w9 AND NOT "Edge_106";   // rising edge
   "Edge_106" := #_w9;
   IF #_w10 THEN "LIFT_3"."Jog+" := TRUE; END_IF;
   #_w11 := NOT #_w9 AND "Edge_107";   // falling edge
   "Edge_107" := #_w9;
   IF #_w11 THEN "LIFT_3"."Jog+" := FALSE; END_IF;
   #_w12 := "MANUAL_STATE" AND "Manual_Jog_BW_Lift3";
   #_w13 := #_w12 AND NOT "Edge_108";   // rising edge
   "Edge_108" := #_w12;
   IF #_w13 THEN "LIFT_3"."Jog-" := TRUE; END_IF;
   #_w14 := NOT #_w12 AND "Edge_109";   // falling edge
   "Edge_109" := #_w12;
   IF #_w14 THEN "LIFT_3"."Jog-" := FALSE; END_IF;
   #_w15 := "MANUAL_STATE" AND "Manual_RUN_FW_Lift3";
   #_w16 := #_w15 AND NOT "Edge_122";   // rising edge
   "Edge_122" := #_w15;
   IF #_w16 THEN "LIFT_3".Run_FW := TRUE; END_IF;
   #_w17 := NOT #_w15 AND "Edge_123";   // falling edge
   "Edge_123" := #_w15;
   IF #_w17 THEN "LIFT_3".Run_FW := FALSE; END_IF;
   #_w18 := "MANUAL_STATE" AND "Manual_RUN_BW_Lift3";
   #_w19 := #_w18 AND NOT "Edge_124";   // rising edge
   "Edge_124" := #_w18;
   IF #_w19 THEN "LIFT_3".Run_BW := TRUE; END_IF;
   #_w20 := NOT #_w18 AND "Edge_125";   // falling edge
   "Edge_125" := #_w18;
   IF #_w20 THEN "LIFT_3".Run_BW := FALSE; END_IF;
END_REGION

REGION Network 24: Input Conveyor
   RUNG wire#powerrail
      Contact( "Run_FW_Conveyor_Input" )
      wire#w1
      I_Contact( "Motor Băng tải Input_2" )
      Coil( "Motor Băng tải Input" )
   END_RUNG
   RUNG wire#powerrail
      Contact( "MANUAL_STATE" )
      Contact( "Manual_Run_FW_Input_Conveyor" )
   END_RUNG wire#w1
   RUNG wire#powerrail
      Contact( "Run_BW_Conveyor_Input" )
      wire#w2
      I_Contact( "Motor Băng tải Input" )
      Coil( "Motor Băng tải Input_2" )
   END_RUNG
   RUNG wire#powerrail
      Contact( "MANUAL_STATE" )
      Contact( "Manual_Run_BW_Input_Conveyor" )
   END_RUNG wire#w2
   // the same network as SCL:
   "Motor Băng tải Input" := ("Run_FW_Conveyor_Input" OR ("MANUAL_STATE" AND "Manual_Run_FW_Input_Conveyor")) AND NOT "Motor Băng tải Input_2";
   "Motor Băng tải Input_2" := ("Run_BW_Conveyor_Input" OR ("MANUAL_STATE" AND "Manual_Run_BW_Input_Conveyor")) AND NOT "Motor Băng tải Input";
END_REGION

REGION Network 25: Output Conveyor
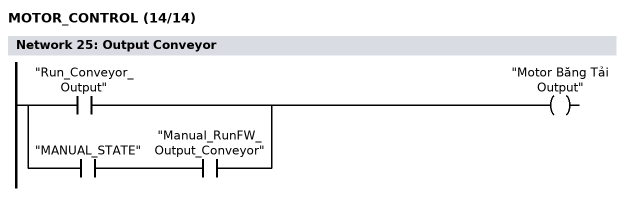
   RUNG wire#powerrail
      Contact( "Run_Conveyor_Output" )
      wire#w1
      Coil( "Motor Băng Tải Output" )
   END_RUNG
   RUNG wire#powerrail
      Contact( "MANUAL_STATE" )
      Contact( "Manual_RunFW_Output_Conveyor" )
   END_RUNG wire#w1
   // the same network as SCL:
   "Motor Băng Tải Output" := "Run_Conveyor_Output" OR ("MANUAL_STATE" AND "Manual_RunFW_Output_Conveyor");
END_REGION
END_ORGANIZATION_BLOCK

ORGANIZATION_BLOCK "TCP_CONTROL"   // OB124, LAD, ProgramCycle
TITLE = "Main Program Sweep (Cycle)"
{ S7_Optimized_Access := 'TRUE' }
VERSION : 0.1
   VAR_INPUT
      Initial_Call : Bool;   // Initial call of this OB
      Remanence : Bool;   // =True, if remanent data are available
   END_VAR
   VAR_TEMP   // added for the SCL form of the ladder/FBD networks
      _w1 : Bool;
      _w2 : Bool;
      _w3 : Bool;
   END_VAR
BEGIN

REGION Network 1: Establish TCP Connection
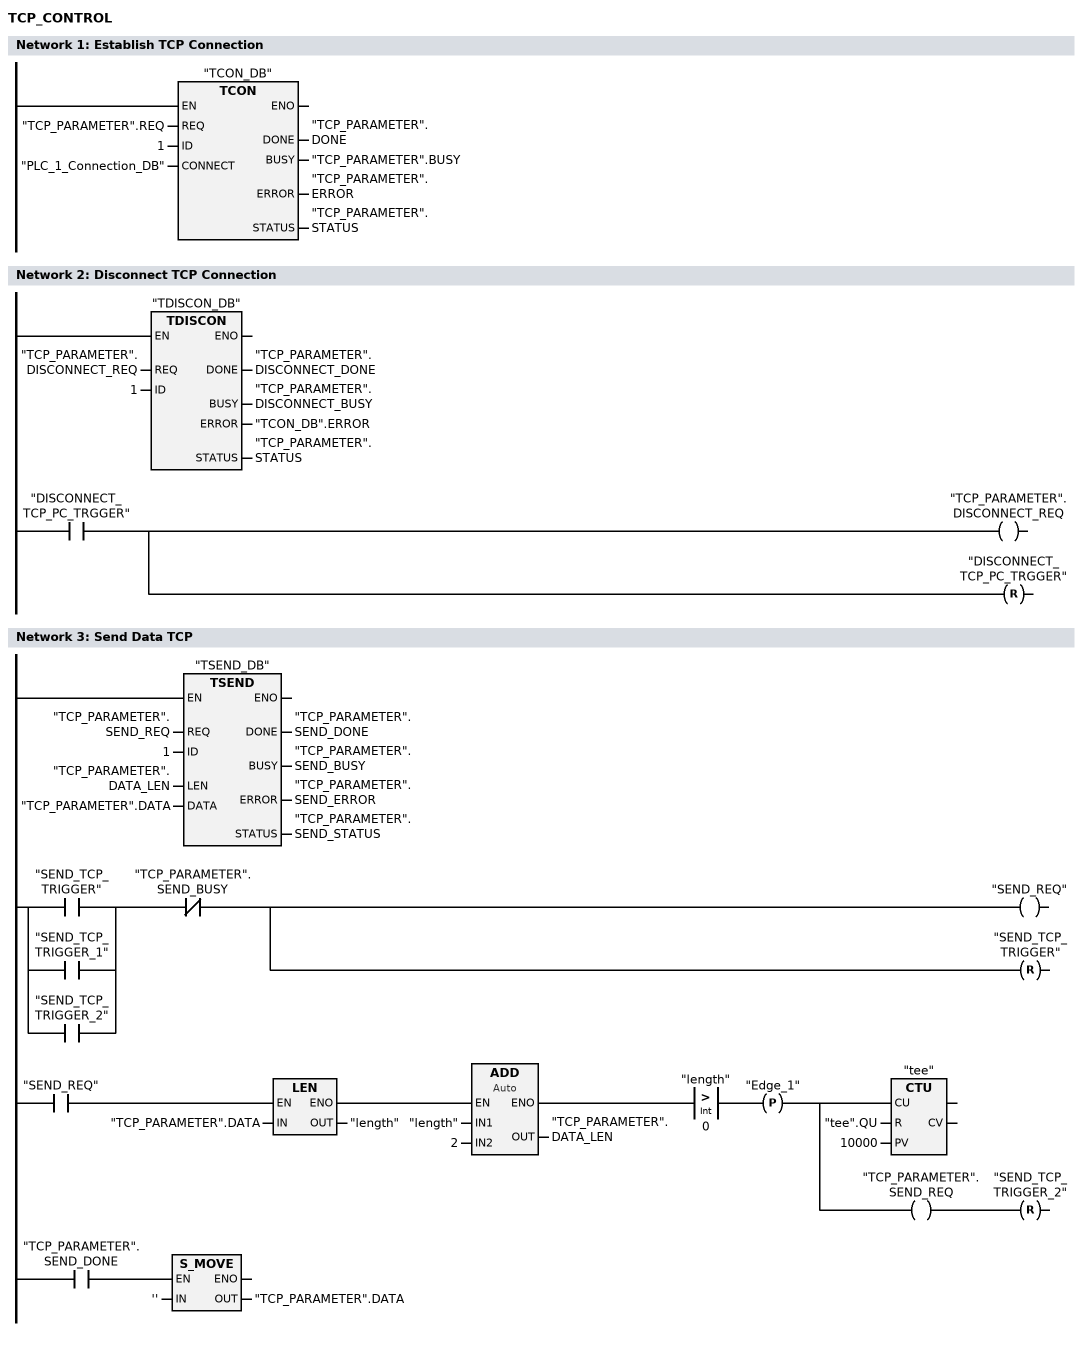
   "TCON_DB"(REQ := "TCP_PARAMETER".REQ,   // TCON
             ID := 1,
             CONNECT := "PLC_1_Connection_DB",
             DONE => "TCP_PARAMETER".DONE,
             BUSY => "TCP_PARAMETER".BUSY,
             ERROR => "TCP_PARAMETER".ERROR,
             STATUS => "TCP_PARAMETER".STATUS);
END_REGION

REGION Network 2: Disconnect TCP Connection
   "TDISCON_DB"(REQ := "TCP_PARAMETER".DISCONNECT_REQ,   // TDISCON
                ID := 1,
                DONE => "TCP_PARAMETER".DISCONNECT_DONE,
                BUSY => "TCP_PARAMETER".DISCONNECT_BUSY,
                ERROR => "TCON_DB".ERROR,
                STATUS => "TCP_PARAMETER".STATUS);
   "TCP_PARAMETER".DISCONNECT_REQ := "DISCONNECT_TCP_PC_TRGGER";
   IF "DISCONNECT_TCP_PC_TRGGER" THEN "DISCONNECT_TCP_PC_TRGGER" := FALSE; END_IF;
END_REGION

REGION Network 3: Send Data TCP
   // ENO of a box is taken as its EN; it also drops when the box reports an error
   "TSEND_DB"(REQ := "TCP_PARAMETER".SEND_REQ,   // TSEND
              ID := 1,
              LEN := "TCP_PARAMETER".DATA_LEN,
              DATA := "TCP_PARAMETER".DATA,
              DONE => "TCP_PARAMETER".SEND_DONE,
              BUSY => "TCP_PARAMETER".SEND_BUSY,
              ERROR => "TCP_PARAMETER".SEND_ERROR,
              STATUS => "TCP_PARAMETER".SEND_STATUS);
   "SEND_REQ" := ("SEND_TCP_TRIGGER" OR "SEND_TCP_TRIGGER_1" OR "SEND_TCP_TRIGGER_2") AND NOT "TCP_PARAMETER".SEND_BUSY;
   IF "SEND_REQ" THEN "SEND_TCP_TRIGGER" := FALSE; END_IF;
   #_w1 := "SEND_REQ";
   IF #_w1 THEN
       "length" := LEN(IN := "TCP_PARAMETER".DATA);
       "TCP_PARAMETER".DATA_LEN := "length" + 2;
   END_IF;
   #_w2 := #_w1 AND ("length" > 0);
   #_w3 := #_w2 AND NOT "Edge_1";   // rising edge
   "Edge_1" := #_w2;
   "tee".CTU(CU := #_w3, R := "tee".QU, PV := 10000);
   "TCP_PARAMETER".SEND_REQ := #_w3;
   IF #_w3 THEN "SEND_TCP_TRIGGER_2" := FALSE; END_IF;
   IF "TCP_PARAMETER".SEND_DONE THEN "TCP_PARAMETER".DATA := ''; END_IF;
END_REGION
END_ORGANIZATION_BLOCK